	        // Check if a Controller has an error
	        #sx_ErrorActive := (#sx_ErrorController AND #iUDT_AixConfig.Motor.MotorExist)
	        OR #sFB_TimerOnOffDelayMCORunningFeedbackError.qx_DelayedSignal
	        OR #sFB_TimerOnOffDelayMCOSpeedFeedbackError.qx_DelayedSignal;

	        // Internal error
	        #sUDT_HMIStatus.InternalError := #sx_AixAvailableControler AND #sx_ErrorController;

	    END_REGION

	END_REGION

	REGION 5 - Check if configuration is ok for commissioning purposes

	    IF (
	        #iUDT_AixConfig.Motor.MotorExist                            // Check only if motor exists
	        AND (#iUDT_AixConfig.Motor.RampUpTime > 0)                  // If ramp up time is greater than 0
	        AND (#iUDT_AixConfig.Motor.RampDownTime > 0)                // and ramp down time is greater than 0
	        )
	        AND
	        (
	        #sUDT_PNDeviceController.PNDeviceFound
	        OR NOT #iUDT_AixConfig.Motor.MotorExist                       // and device found in PN structure
	        OR #ix_SimulationModeActive                                 // or simulation mode is active
	        )
	    THEN
	        #sx_ConfigurationError := FALSE;                                // Reset configuration error
	    ELSE
	        #sx_ConfigurationError := TRUE;                                 // Set configuration error
	    END_IF;

	END_REGION

	REGION 6 - Prepare output data for Controller

	    REGION 6.1 - Set direction for motor

	        // If Run forward is requested, set direction to forward
	        IF #iqUDT_ConveyorInterface.RunFwd
	            AND #iUDT_AixConfig.Motor.InterlockFwd
	        THEN
	            #sx_RunForward := TRUE;
	            #sx_RunReverse := FALSE;
	        END_IF;

	        // If Run reverse is requested, set direction into reverse
	        IF #iqUDT_ConveyorInterface.RunRvs
	            AND #iUDT_AixConfig.Motor.InterlockRvs
	        THEN
	            #sx_RunReverse := TRUE;
	            #sx_RunForward := FALSE;
	        END_IF;

	    END_REGION


	    REGION 6.3 - Stopping motor

	        // Create trigger when direction signal falling
	        #sF_TRIG_RunFwd(CLK := #iqUDT_ConveyorInterface.RunFwd);
	        #sF_TRIG_RunRvs(CLK := #iqUDT_ConveyorInterface.RunRvs);

	        // When no run signal is given the controllers should stop
	        IF (NOT #iqUDT_ConveyorInterface.RunRvs AND NOT #iqUDT_ConveyorInterface.RunFwd)
	            OR (#iqUDT_ConveyorInterface.RunRvs AND #iqUDT_ConveyorInterface.RunFwd)
	            OR (#sF_TRIG_RunRvs.Q)
	            OR (#sF_TRIG_RunFwd.Q)
	            OR #sx_ErrorActive
	        THEN
	            #sx_RunReverse := FALSE;
	            #sx_RunForward := FALSE;
	        END_IF;

	    END_REGION

	    REGION 6.5 - Check for enable operation signal

	        //Enable operation if there is no error active and there is an given direction
	        #sx_EnableOperation := NOT #sx_ErrorActive
	        AND NOT #sx_ConfigurationError
	        AND (#sx_RunForward OR #sx_RunReverse);
	    END_REGION

	    REGION 6.6 - Calculate acceleration and deceleration values

	        //Motor
	        //Recalculating Acceleration (from ms to mm)
	        #si_MotorAcceleration := REAL_TO_INT((INT_TO_REAL(#iqUDT_ConveyorInterface.SpeedSetpoint) * #iUDT_AixConfig.Motor.Ratio / 2) * (UDINT_TO_REAL(#iUDT_AixConfig.Motor.RampUpTime) / 1000));

	        //Recalculating Deceleration (from ms to mm)
	        #si_MotorDeceleration := REAL_TO_INT((INT_TO_REAL(#iqUDT_ConveyorInterface.SpeedSetpoint) * #iUDT_AixConfig.Motor.Ratio / 2) * (UDINT_TO_REAL(#iUDT_AixConfig.Motor.RampDownTime) / 1000));

	    END_REGION

	END_REGION

	REGION 7 - Write outputs to controller
	    // Clear speed setpoint when no run request or above direction request or is configuration error
	    IF #sx_EnableOperation
	    THEN
	        #sr_ActualSpeedSetpoint := INT_TO_REAL(#iqUDT_ConveyorInterface.SpeedSetpoint) / #iUDT_AixConfig.Motor.Ratio;
	    ELSE
	        #sr_ActualSpeedSetpoint := 0;
	    END_IF;

	    REGION 7.1 - Controller Left motor

	        IF #ii_MotorPositionId = #ci_Master_Left OR #ii_MotorPositionId = #ci_Slave_Left THEN
	            //Seting up speed for Left motor
	            #iqUDT_AixOutputsModule.LeftSetMotorSpeed := REAL_TO_INT(#sr_ActualSpeedSetpoint);
	            IF #iqUDT_AixOutputsModule.LeftSetMotorSpeed > #cr_MaximumOutput
	            THEN
	                // if actual value is greater than maximmu output value then write maximmu output value
	                #iqUDT_AixOutputsModule.LeftSetMotorSpeed := REAL_TO_INT(#cr_MaximumOutput);
	            END_IF;

	            //Check if motor is in use, if yes set parameters from conveyor to the controller and motor
	            IF #iUDT_AixConfig.Motor.MotorExist
	            THEN
	                //Setting up run bit, acceleration, deceleration
	                #iqUDT_AixOutputsModule.LeftMotorControl.Run := #sx_EnableOperation
	                AND (#iqUDT_ConveyorInterface.RunFwd OR #iqUDT_ConveyorInterface.RunRvs);

	                // Position setpoint
	                #iqUDT_AixOutputsModule.ServoControlDistanceLeft := #ii_PositionSetpoint;

	                //Start positioning
	                #iqUDT_AixOutputsModule.ServoControlCommandLeft.%X1 := #ix_StartPositioning
	                AND #sx_EnableOperation
	                AND (#iqUDT_ConveyorInterface.RunFwd OR #iqUDT_ConveyorInterface.RunRvs);

	                // Reset position
	                #sR_TRIG_ResetPosition(CLK := #ix_ResetPosition);

	                // Reset position after every operation
	                IF #sR_TRIG_ResetPosition.Q THEN

	                    #iqUDT_AixOutputsModule.ServoControlCommandLeft.%X0 := TRUE;

	                END_IF;

	                // End homing procedure when motor is reset
	                IF #iUDT_AixInputsModule.ServoStatusLeft.%X1 THEN

	                    #iqUDT_AixOutputsModule.ServoControlCommandLeft.%X0 := FALSE;

	                END_IF;


	                #iqUDT_AixOutputsModule.LeftSetMotorAccel := #si_MotorAcceleration;
	                #iqUDT_AixOutputsModule.LeftSetMotorDeccel := #si_MotorDeceleration;

	                //Setting direction
	                IF (#sx_RunReverse AND NOT #iUDT_AixConfig.Motor.DirectionReversal)
	                    OR (#sx_RunForward AND #iUDT_AixConfig.Motor.DirectionReversal)
	                THEN
	                    #iqUDT_AixOutputsModule.LeftMotorControl.MotorDirection := 1;
	                ELSE
	                    #iqUDT_AixOutputsModule.LeftMotorControl.MotorDirection := 0;
	                END_IF;
	            ELSE
	                #iqUDT_AixOutputsModule.LeftMotorControl.Run := FALSE;
	            END_IF;
	        END_IF;
	    END_REGION

	    REGION 7.2 - Controller right motor
	        IF #ii_MotorPositionId = #ci_Master_Right OR #ii_MotorPositionId = #ci_Slave_Right THEN
	            //Seting up speed for Right motor
	            #iqUDT_AixOutputsModule.RightSetMotorSpeed := REAL_TO_INT(#sr_ActualSpeedSetpoint);
	            IF #iqUDT_AixOutputsModule.RightSetMotorSpeed > #cr_MaximumOutput
	            THEN
	                // if actual value is greater than maximmu output value then write maximmu output value
	                #iqUDT_AixOutputsModule.RightSetMotorSpeed := REAL_TO_INT(#cr_MaximumOutput);
	            END_IF;

	            //Check if motor is in use, if yes set parameters from conveyor to the controller and motor
	            IF #iUDT_AixConfig.Motor.MotorExist
	            THEN
	                //Setting up run bit, acceleration, deceleration
	                #iqUDT_AixOutputsModule.RightMotorControl.Run := #sx_EnableOperation
	                AND (#iqUDT_ConveyorInterface.RunFwd OR #iqUDT_ConveyorInterface.RunRvs);

	                // Position setpoint
	                #iqUDT_AixOutputsModule.ServoControlDistanceRight := #ii_PositionSetpoint;

	                //Start positioning
	                #iqUDT_AixOutputsModule.ServoControlCommandRight.%X1 := #ix_StartPositioning
	                AND #sx_EnableOperation
	                AND (#iqUDT_ConveyorInterface.RunFwd OR #iqUDT_ConveyorInterface.RunRvs);

	                // Reset position
	                #sR_TRIG_ResetPosition(CLK := #ix_ResetPosition);

	                // Reset position after every operation
	                IF #sR_TRIG_ResetPosition.Q THEN

	                    #iqUDT_AixOutputsModule.ServoControlCommandRight.%X0 := TRUE;

	                END_IF;

	                // End homing procedure when motor is reset
	                IF #iUDT_AixInputsModule.ServoStatusRight.%X1 THEN

	                    #iqUDT_AixOutputsModule.ServoControlCommandRight.%X0 := FALSE;

	                END_IF;


	                #iqUDT_AixOutputsModule.RightSetMotorAccel := #si_MotorAcceleration;
	                #iqUDT_AixOutputsModule.RightSetMotorDeccel := #si_MotorDeceleration;

	                //Setting direction
	                IF (#sx_RunReverse AND NOT #iUDT_AixConfig.Motor.DirectionReversal)
	                    OR (#sx_RunForward AND #iUDT_AixConfig.Motor.DirectionReversal)
	                THEN
	                    #iqUDT_AixOutputsModule.RightMotorControl.MotorDirection := 1;
	                ELSE
	                    #iqUDT_AixOutputsModule.RightMotorControl.MotorDirection := 0;
	                END_IF;
	            ELSE
	                #iqUDT_AixOutputsModule.RightMotorControl.Run := FALSE;
	            END_IF;
	        END_IF;
	    END_REGION

	END_REGION

	REGION 8 - Reading actual speed

	    REGION 8.1 - Left Motor
	        IF #ii_MotorPositionId = #ci_Master_Left OR #ii_MotorPositionId = #ci_Slave_Left THEN
	            //When motors are in constant speed use motor actual speed
	            IF #iUDT_AixConfig.Motor.MotorExist
	            THEN
	                #si_ActualSpeed := REAL_TO_INT(INT_TO_REAL(WORD_TO_INT(#iUDT_AixInputsModule.LeftMotorActualSpeed & #cw_ActualSpeedMask)) * #iUDT_AixConfig.Motor.Ratio);
	            ELSE
	                #si_ActualSpeed := 0;
	            END_IF;
	        END_IF;
	    END_REGION

	    REGION 8.2 - Right Motor
	        IF #ii_MotorPositionId = #ci_Master_Right OR #ii_MotorPositionId = #ci_Slave_Right THEN
	            //When motors are in constant speed use motor actual speed
	            IF #iUDT_AixConfig.Motor.MotorExist
	            THEN
	                #si_ActualSpeed := REAL_TO_INT(INT_TO_REAL(WORD_TO_INT(#iUDT_AixInputsModule.RightMotorActualSpeed & #cw_ActualSpeedMask)) * #iUDT_AixConfig.Motor.Ratio);
	            ELSE
	                #si_ActualSpeed := 0;
	            END_IF;
	        END_IF;
	    END_REGION

	    REGION 8.3 - Calculation
	        //Actual speed is in mm/s
	        //Sets error signal if an motor is running for a longer time with a diferent speed than speed setpoint but after a certain time
	        #sFB_TimerOnOffDelayMCORunningFeedbackError(iudi_OnDelayTime := #cudi_FeedbackErrorDelay,
	                                                    ix_SignalToDelay := #sr_ActualSpeedSetpoint <> 0.0 AND NOT (#si_ActualSpeed <> 0));

	        //The motor should start running after specific time. If not the MCORunningFeedback error occured
	        #sFB_TimerOnOffDelayMCOSpeedFeedbackError(iudi_OnDelayTime := #cudi_FeedbackErrorDelay,
	                                                  ix_SignalToDelay := #sx_SpeedFeedbackError);

	        IF #sFB_TimerOnOffDelayMCORunningFeedbackError.qx_DelayedSignal OR #sFB_TimerOnOffDelayMCOSpeedFeedbackError.qx_DelayedSignal
	        THEN
	            #sUDT_HMIStatus.SpeedFeedbackError := TRUE;
	        END_IF;

	        //Sets signal for the time in which the motors are accelerating
	        #sFB_TimerOnOffDelayAcceleration(iudi_OnDelayTime := 0,
	                                         iudi_OffDelayTime := #iUDT_AixConfig.Motor.RampUpTime + #cudi_TimeOffsetSpeedmonitoring,
	                                         ix_SignalToDelay := #sR_TRIG_Running.Q,
	                                         ix_Enable := TRUE,
	                                         qx_DelayedSignal => #sx_Accelerating);


	        //If conveyor is running and runs forwad or backwards and is not accelerating, when any motor is running at a lower/greater speed than set speed then set an error
	        IF #iqUDT_ConveyorInterface.VFDRunning AND (#iqUDT_ConveyorInterface.RunFwd OR #iqUDT_ConveyorInterface.RunRvs) AND NOT #sx_Accelerating
	        THEN
	            //Check if the difference betwen acctual speed and set speed is bigger than deviation then set error
	            #sx_SpeedFeedbackError := #iUDT_AixConfig.Motor.SpeedSetpointWindow < (ABS(#si_ActualSpeed) - (#iqUDT_ConveyorInterface.SpeedSetpoint));
	        END_IF;


	        // Check IF speed setpoint is reached FOR motor
	        #sx_SpeedSetpointReached := (ABS(#si_ActualSpeed) >= ((#iqUDT_ConveyorInterface.SpeedSetpoint) - #iUDT_AixConfig.Motor.SpeedSetpointWindow))
	        AND (ABS(#si_ActualSpeed) <= ((#iqUDT_ConveyorInterface.SpeedSetpoint) + #iUDT_AixConfig.Motor.SpeedSetpointWindow));
	    END_REGION

	END_REGION

	(* REGION 9 - Reading actual position

	    REGION 9.1 - Left Motor

	        #sx_LeftServoHomeHasBeenSet := #iUDT_AixInputsModule.ServoStatusLeft.%X1;
	        IF #ix_MotorPositionId = #ci_Left
	        THEN
	            IF #sx_LeftServoHomeHasBeenSet THEN
	                #si_LastLeftMotorPosition := 0;
	            END_IF;
	            // Add last position change to static memory
	            #si_LeftMotorPosition += - #si_LastLeftMotorPosition;
	            // Save last motor position
	            #si_LastLeftMotorPosition := #iUDT_AixInputsModule.ServoLocationLeft;

	            // Copy displacement if motor position change is greater or equal to 1 cm and store rest
	            IF #si_LeftMotorPosition > 10 THEN
	                #iqUDT_ConveyorInterface.DeltaPosition := REAL_TO_INT(INT_TO_REAL(#si_LeftMotorPosition) * #iUDT_AixConfig.Motor.Ratio) / 10;
	                #si_LeftMotorPosition := #si_LeftMotorPosition MOD 10;
	            ELSE
	                #iqUDT_ConveyorInterface.DeltaPosition := 0;
	            END_IF;

	            // allocate Motor Rotation status
	            #sb_MotorRotationStatus.%X0 := #iUDT_AixInputsModule.LeftMotorDiagnostic.MotorStatus1;
	            #sb_MotorRotationStatus.%X1 := #iUDT_AixInputsModule.LeftMotorDiagnostic.MotorStatus2;

	            // Change direction sign if motor running reverse
	            IF ((#sb_MotorRotationStatus = #cb_MotorInCW) AND NOT #iUDT_AixConfig.Motor.DirectionReversal) OR
	                ((#sb_MotorRotationStatus = #cb_MotorInCCW) AND #iUDT_AixConfig.Motor.DirectionReversal)
	            THEN

	                #iqUDT_ConveyorInterface.DeltaPosition *= -1;

	            END_IF;

	            // Motor positioned
	            #qx_Positioned := #iUDT_AixInputsModule.ServoStatusLeft.%X0;

	        END_IF;

	    END_REGION

	    REGION 9.2 - Right motor
	        #sx_RightServoHomeHasBeenSet := #iUDT_AixInputsModule.ServoStatusRight.%X1;
	        IF #ix_MotorPositionId = #ci_Right
	        THEN
	            IF #sx_RightServoHomeHasBeenSet THEN
	                #si_LastRightMotorPosition := 0;
	            END_IF;
	            // Add last position change to static memory
	            #si_RightMotorPosition += - #si_LastRightMotorPosition;
	            // Save last motor position
	            #si_LastRightMotorPosition := #iUDT_AixInputsModule.ServoLocationRight;

	            // Copy displacement if motor position change is greater or equal to 1 cm and store rest
	            IF #si_RightMotorPosition > 10 THEN
	                #iqUDT_ConveyorInterface.DeltaPosition := REAL_TO_INT(INT_TO_REAL(#si_RightMotorPosition) * #iUDT_AixConfig.Motor.Ratio) / 10;
	                #si_RightMotorPosition := #si_RightMotorPosition MOD 10;
	            ELSE
	                #iqUDT_ConveyorInterface.DeltaPosition := 0;
	            END_IF;

	            // allocate Motor Rotation status
	            #sb_MotorRotationStatus.%X0 := #iUDT_AixInputsModule.RightMotorDiagnostic.MotorStatus1;
	            #sb_MotorRotationStatus.%X1 := #iUDT_AixInputsModule.RightMotorDiagnostic.MotorStatus2;

	            // Change direction sign if motor running reverse
	            IF ((#sb_MotorRotationStatus = #cb_MotorInCW) AND NOT #iUDT_AixConfig.Motor.DirectionReversal) OR
	                ((#sb_MotorRotationStatus = #cb_MotorInCCW) AND #iUDT_AixConfig.Motor.DirectionReversal)
	            THEN

	                #iqUDT_ConveyorInterface.DeltaPosition *= -1;

	            END_IF;

	            // Motor positioned
	            #qx_Positioned := #iUDT_AixInputsModule.ServoStatusRight.%X0;

	        END_IF;

	    END_REGION


	END_REGION *)

	REGION 9 - Reading actual position

	    REGION 9.1 - Left motor

	        IF #ii_MotorPositionId = #ci_Master_Left OR #ii_MotorPositionId = #ci_Slave_Left
	        THEN
	            IF #iUDT_AixInputsModule.ServoLocationLeft = 0 THEN
	                #si_LastLeftMotorPosition := 0;
	            END_IF;
	            // Add last position change to static memory
	            #si_LeftMotorPosition += ABS(ABS(#iUDT_AixInputsModule.ServoLocationLeft) - ABS(#si_LastLeftMotorPosition));
	            // Save last motor position
	            #si_LastLeftMotorPosition := #iUDT_AixInputsModule.ServoLocationLeft;

	            // Copy delta position if motor position change is greater or equal to 1 cm and store rest
	            IF #si_LeftMotorPosition > 10 THEN
	                IF #ii_MotorPositionId = #ci_Master_Left THEN
	                    #iqUDT_ConveyorInterface.DeltaPosition := REAL_TO_INT(INT_TO_REAL(#si_LeftMotorPosition) * #iUDT_AixConfig.Motor.Ratio) / 10;
	                END_IF;
	                #si_LeftMotorPosition := #si_LeftMotorPosition MOD 10;
	            ELSE
	                IF #ii_MotorPositionId = #ci_Master_Left THEN
	                    #iqUDT_ConveyorInterface.DeltaPosition := 0;
	                END_IF;
	            END_IF;
	            // Change direction sign if motor running reverse
	            IF #iUDT_AixInputsModule.LeftMotorDiagnostic.MotorStatus1 AND NOT #iUDT_AixInputsModule.LeftMotorDiagnostic.MotorStatus2 AND NOT #iUDT_AixConfig.Motor.DirectionReversal
	                OR NOT #iUDT_AixInputsModule.LeftMotorDiagnostic.MotorStatus1 AND #iUDT_AixInputsModule.LeftMotorDiagnostic.MotorStatus2 AND #iUDT_AixConfig.Motor.DirectionReversal
	            THEN
	                IF #ii_MotorPositionId = #ci_Master_Left THEN
	                    #iqUDT_ConveyorInterface.DeltaPosition *= -1;
	                END_IF;
	            END_IF;

	            // Motor positioned
	            #qx_Positioned := #iUDT_AixInputsModule.ServoStatusLeft.%X0;

	        END_IF;

	    END_REGION

	    REGION 9.2 - Right motor

	        IF #ii_MotorPositionId = #ci_Master_Right OR #ii_MotorPositionId = #ci_Slave_Right
	        THEN
	            IF #iUDT_AixInputsModule.ServoLocationRight = 0 THEN
	                #si_LastRightMotorPosition := 0;
	            END_IF;
	            // Add last position change to static memory
	            #si_RightMotorPosition += ABS(ABS(#iUDT_AixInputsModule.ServoLocationRight) - ABS(#si_LastRightMotorPosition));
	            // Save last motor position
	            #si_LastRightMotorPosition := #iUDT_AixInputsModule.ServoLocationRight;

	            // Copy delta position if motor position change is greater or equal to 1 cm and store rest
	            IF #si_RightMotorPosition > 10 THEN
	                IF #ii_MotorPositionId = #ci_Master_Right THEN
	                    #iqUDT_ConveyorInterface.DeltaPosition := REAL_TO_INT(INT_TO_REAL(#si_RightMotorPosition) * #iUDT_AixConfig.Motor.Ratio) / 10;
	                END_IF;
	                #si_RightMotorPosition := #si_RightMotorPosition MOD 10;
	            ELSE
	                IF #ii_MotorPositionId = #ci_Master_Right THEN
	                    #iqUDT_ConveyorInterface.DeltaPosition := 0;
	                END_IF;
	            END_IF;
	            // Change direction sign if motor running reverse
	            IF #iUDT_AixInputsModule.RightMotorDiagnostic.MotorStatus1 AND NOT #iUDT_AixInputsModule.RightMotorDiagnostic.MotorStatus2 AND NOT #iUDT_AixConfig.Motor.DirectionReversal
	                OR NOT #iUDT_AixInputsModule.RightMotorDiagnostic.MotorStatus1 AND #iUDT_AixInputsModule.RightMotorDiagnostic.MotorStatus2 AND #iUDT_AixConfig.Motor.DirectionReversal
	            THEN
	                IF #ii_MotorPositionId = #ci_Master_Right THEN
	                    #iqUDT_ConveyorInterface.DeltaPosition *= -1;
	                END_IF;
	            END_IF;

	            // Motor positioned
	            #qx_Positioned := #iUDT_AixInputsModule.ServoStatusRight.%X0;

	        END_IF;

	    END_REGION

	END_REGION


	REGION 10 - Copy signals to interface DB and to status output UDT

	    REGION 10.1 - Motor

	        // Create internal error status
	        // Write Conveyor interface bits only if it is a Master
	        IF #ii_MotorPositionId = #ci_Master_Left OR #ii_MotorPositionId = #ci_Master_Right THEN

	            #iqUDT_ConveyorInterface.VFDRunning := #sx_AixAvailableControler AND
	            (#si_ActualSpeed <> 0);                 // Write true on output Conveyor interface structure if Ai2's are in operation and motor is turning

	            #iqUDT_ConveyorInterface.VFDatSpeed := #sx_SpeedSetpointReached AND
	            #sx_AixAvailableControler AND
	            #si_ActualSpeed <> 0 AND
	            NOT #sx_SpeedFeedbackError;             // Copy setpoint speed reached state from static to the output conveyor interface structure

	            #iqUDT_ConveyorInterface.InternalWarningVFD := #sUDT_HMIStatus.PNSlaveWarning;                                                       // Set the internal warning bit if any warning is active

	            #iqUDT_ConveyorInterface.InternalErrorVFD := #sx_ErrorCMotor;                   // Set the internal error bit if any fault is active

	            #iqUDT_ConveyorInterface.ActualSpeed := ABS(#si_ActualSpeed);                   // Copy the calculated value to the output

	            #iqUDT_ConveyorInterface.ConfigurationError := #sx_ConfigurationError;          // Copy the calculated value to the output

	        END_IF;


	    END_REGION

	    REGION 10.2 - Move error status TO HMI Status

	        // Copy error status to output
	        #qUDT_HMIStatus := #sUDT_HMIStatus;

	    END_REGION

	END_REGION

	REGION 11 - Statistic

	    REGION 11.1 - General
	        // Statement section REGION
	        #sx_GeneralStatisticsReset := #iqUDT_ConveyorInterface.ResetStatistics;
	    END_REGION

	    // Create trigger on error and create statistics for profinet slave not online
	    #sR_TRIG_PNSlaveNotOnline(CLK := #sUDT_HMIStatus.PNSlaveNotOnline);                 // Detect the rising edge of the error

	    IF #sx_GeneralStatisticsReset OR #sUDT_HMIStatus.PNSlaveNotOnline
	    THEN

	        "FC_Statistics"(ix_Reset := #sx_GeneralStatisticsReset,
	                        ix_Activate := #sUDT_HMIStatus.PNSlaveNotOnline,
	                        ix_RTrigActivate := #sR_TRIG_PNSlaveNotOnline.Q,
	                        iqUDT_Statistics := #iqUDT_MCOStatistics.PNSlaveNotOnline);

	        #iqUDT_MCOStatistics.PNSlaveNotOnline := #iqUDT_MCOStatistics.PNSlaveNotOnline;
	    END_IF;

	    // Create trigger on error and create statistics for profinet slave error
	    #sR_TRIG_PNSlaveError(CLK := #sUDT_HMIStatus.PNSlaveError);                                                                          // Detect the rising edge of the error

	    IF #sx_GeneralStatisticsReset OR #sUDT_HMIStatus.PNSlaveError
	    THEN

	        "FC_Statistics"(ix_Reset := #sx_GeneralStatisticsReset,
	                        ix_Activate := #sUDT_HMIStatus.PNSlaveError,
	                        ix_RTrigActivate := #sR_TRIG_PNSlaveError.Q,
	                        iqUDT_Statistics := #iqUDT_MCOStatistics.PNSlaveError);

	        #iqUDT_MCOStatistics.PNSlaveError := #iqUDT_MCOStatistics.PNSlaveError;
	    END_IF;


	    // Create trigger on error and create statistics for MCO communication error
	    #sR_TRIG_CommunicationErrorMCO(CLK := #qUDT_HMIStatus.CommunicationErrorVFD);            // Detect the rising edge of the error

	    IF #sx_GeneralStatisticsReset OR #qUDT_HMIStatus.CommunicationErrorVFD
	    THEN

	        "FC_Statistics"(ix_Reset := #sx_GeneralStatisticsReset,
	                        ix_Activate := #qUDT_HMIStatus.CommunicationErrorVFD,
	                        ix_RTrigActivate := #sR_TRIG_CommunicationErrorMCO.Q,
	                        iqUDT_Statistics := #iqUDT_MCOStatistics.CommunicationErrorMovikit);

	    END_IF;

	    REGION 11.1 - Motor

	        // Create trigger on error and create statistics for internal MCO Error
	        #sR_TRIG_MCOInternalError(CLK := #sUDT_HMIStatus.InternalError);         // Detect the rising edge of the error

	        IF #iqUDT_ConveyorInterface.ResetStatistics OR #sUDT_HMIStatus.InternalError
	        THEN

	            "FC_Statistics"(ix_Reset := #iqUDT_ConveyorInterface.ResetStatistics,
	                            ix_Activate := #sUDT_HMIStatus.InternalError,
	                            ix_RTrigActivate := #sR_TRIG_MCOInternalError.Q,
	                            iqUDT_Statistics := #iqUDT_MCOStatistics.VFDInternalError);

	        END_IF;

	        // Create trigger on running signal and create statistics for running status
	        #sR_TRIG_Running(CLK := #iqUDT_ConveyorInterface.VFDRunning);                           // Detect the rising edge of the signal

	        IF #iqUDT_ConveyorInterface.ResetStatistics OR #iqUDT_ConveyorInterface.VFDRunning
	        THEN

	            "FC_Statistics"(ix_Reset := #iqUDT_ConveyorInterface.ResetStatistics,
	                            ix_Activate := #iqUDT_ConveyorInterface.VFDRunning,
	                            ix_RTrigActivate := #sR_TRIG_Running.Q,
	                            iqUDT_Statistics := #iqUDT_MCOStatistics.Running);
	        END_IF;


	    END_REGION
	    REGION 12 Status bit allocation
	        "FC_BitAllocation"(ix_Bit0 := #qUDT_HMIStatus.SpeedFeedbackError,
	                           ix_Bit1 := #qUDT_HMIStatus.InternalWarning,
	                           ix_Bit2 := #qUDT_HMIStatus.InternalError,
	                           ix_Bit3 := #qUDT_HMIStatus.CommunicationErrorVFD,
	                           ix_Bit4 := #qUDT_HMIStatus.PNSlaveNotOnline,
	                           ix_Bit5 := #qUDT_HMIStatus.PNSlaveError,
	                           ix_Bit6 := #qUDT_HMIStatus.PNSlaveWarning,
	                           ix_Bit7 := FALSE,
	                           ix_Bit8 := FALSE,
	                           ix_Bit9 := FALSE,
	                           ix_Bit10 := FALSE,
	                           ix_Bit11 := FALSE,
	                           ix_Bit12 := FALSE,
	                           ix_Bit13 := FALSE,
	                           ix_Bit14 := FALSE,
	                           ix_Bit15 := FALSE,
	                           ix_Bit16 := FALSE,
	                           ix_Bit17 := FALSE,
	                           ix_Bit18 := FALSE,
	                           ix_Bit19 := FALSE,
	                           ix_Bit20 := FALSE,
	                           ix_Bit21 := FALSE,
	                           ix_Bit22 := FALSE,
	                           ix_Bit23 := FALSE,
	                           ix_Bit24 := FALSE,
	                           ix_Bit25 := FALSE,
	                           ix_Bit26 := FALSE,
	                           ix_Bit27 := FALSE,
	                           ix_Bit28 := FALSE,
	                           ix_Bit29 := FALSE,
	                           ix_Bit30 := FALSE,
	                           ix_Bit31 := FALSE,
	                           qdw_Dword => #qUDT_HMIStatus.ControllerStatus);
	    END_REGION
	END_REGION
END_FUNCTION_BLOCK

FUNCTION_BLOCK "FB_Displacement"
TITLE = FB_Displacement
{ S7_Optimized_Access := 'TRUE' }
AUTHOR : MHSE
FAMILY : GeneralSystemFunctions
VERSION : 3.0
//Function block to calculate the displacement.
   VAR_IN_OUT
      iqUDT_ConveyorInterface : "UDT_ConveyorInterface";   // Conveyor interface structure Motor
   END_VAR

   VAR
      slr_FormDisplacement { ExternalAccessible := 'False'; ExternalVisible := 'False'; ExternalWritable := 'False'} : LReal;   // Conveyor displacement [cm]
      slr_Correction { ExternalAccessible := 'False'; ExternalVisible := 'False'; ExternalWritable := 'False'} : LReal;   // Correction [cm]
      sx_PositionModeActive { ExternalAccessible := 'False'; ExternalVisible := 'False'; ExternalWritable := 'False'} : Bool;   // Position Mode is used, Will reset after power change
   END_VAR

   VAR_TEMP
      ti_Displacement : Int;   // Conveyor displacement [cm]
   END_VAR

   VAR CONSTANT
      ci_IntMin : Int := -32768;
      ci_IntMax : Int := 32767;
   END_VAR


BEGIN
	(*
	----------------------------------------------------------------------------------------

	Version history:
	Date        | Version   | Author        | Remark
	----------------------------------------------------------------------------------------
	24/05/2019  | 0.1       | L.Klar        | first release MHS TIA 15.1
	24/07/2019  | 2.0       | L.Klar        | 2.0 MHS library release TIA 15.1
	12/09/2019  | 2.1       | P.Majka       | Comments updataed
	04/11/2019  | 2.2       | L.Klar        | Prevoius cycle scan changed from memory to DB variable
	12/11/2019  | 3.0       | P.Majka       | 3.0 MHS library release TIA 15.1
	21/02/2023  | 4.0       | F.Baten       | 4.0 Release TIA 17.5
	31/05/2024  | 4.1       | I.Ajram       | Added Displacement from Position feedback
	*)
	REGION 0 - Mode detection
	    IF #iqUDT_ConveyorInterface.DeltaPosition <> 0 THEN
	        #sx_PositionModeActive := true;
	    END_IF;
	END_REGION


	REGION 1 - Displacement From Speed
	    IF NOT #sx_PositionModeActive THEN
	        REGION 1.1 Calculate Displacement
	            // Displacement is calculated using actual conveyor speed and the previous PLC cycle scan time
	            #slr_FormDisplacement := INT_TO_LREAL(#iqUDT_ConveyorInterface.ActualSpeed) * "DB_Memory".PrevCycleTime / 10000.0;

	            // Correction is used to accumulate the rest of the calculated value
	            #slr_Correction := FRAC(#slr_FormDisplacement) + #slr_Correction;

	            // The actual displacement is a sum of complete parts of the displacement and correction variables
	            #ti_Displacement := DINT_TO_INT(TRUNC(#slr_FormDisplacement) + TRUNC(#slr_Correction));

	        END_REGION

	        REGION 1.2 - Correction check

	            // Correction incrementation or decremantation if it exceeds 1 or -1 in case of negative speed
	            IF (#slr_Correction >= 1)
	            THEN

	                #slr_Correction -= 1;

	            ELSIF (#slr_Correction <= -1)
	            THEN

	                #slr_Correction += 1;

	            END_IF;

	        END_REGION

	        #iqUDT_ConveyorInterface.Displacement := #ti_Displacement;
	    END_IF;
	END_REGION

	REGION 2 - Displacement from Position
	    // pass position displacement from Servo Feedback
	    IF #sx_PositionModeActive THEN
	        #iqUDT_ConveyorInterface.Displacement := #iqUDT_ConveyorInterface.DeltaPosition;

	    END_IF;

	END_REGION
END_FUNCTION_BLOCK

FUNCTION_BLOCK "FB_RightAngledTransfer"
{ S7_Optimized_Access := 'TRUE' }
VERSION : 0.1
   VAR_INPUT
      iUDT_Configuration { ExternalAccessible := 'False'; ExternalVisible := 'False'; ExternalWritable := 'False'} : "UDT_RATConfiguration" := ((), (), (), (), (), (), (), (), (), (), (), (), (), (), 1, 2, 3, 4, (), (), (), ());   // Configuration structure
      iUDT_LowerConveyorConfiguration { ExternalAccessible := 'False'; ExternalVisible := 'False'; ExternalWritable := 'False'} : "UDT_ConveyorConfiguration";   // Lower configuration structure
      iUDT_UpperConveyorConfiguration { ExternalAccessible := 'False'; ExternalVisible := 'False'; ExternalWritable := 'False'} : "UDT_ConveyorConfiguration";   // Upper configuration structure
      iUDT_PECConfiguration { ExternalAccessible := 'False'; ExternalVisible := 'False'; ExternalWritable := 'False'} : "UDT_PECConfiguration";   // PEC configuration structure
      ii_DestinationA { ExternalAccessible := 'False'; ExternalVisible := 'False'; ExternalWritable := 'False'} : Int;   // Forced destination for every product from conveyor A. When this is 0 then destination is taken from GIN
      ii_DestinationB { ExternalAccessible := 'False'; ExternalVisible := 'False'; ExternalWritable := 'False'} : Int;   // Forced destination for every product from conveyor B. When this is 0 then destination is taken from GIN
      ii_DestinationC { ExternalAccessible := 'False'; ExternalVisible := 'False'; ExternalWritable := 'False'} : Int;   // Forced destination for every product from conveyor C. When this is 0 then destination is taken from GIN
      ii_DestinationD { ExternalAccessible := 'False'; ExternalVisible := 'False'; ExternalWritable := 'False'} : Int;   // Forced destination for every product from conveyor D. When this is 0 then destination is taken from GIN
      ix_HardwareOk { ExternalAccessible := 'False'; ExternalVisible := 'False'; ExternalWritable := 'False'} : Bool;   // TRUE when  hardware is Ok
      ix_400vOk { ExternalAccessible := 'False'; ExternalVisible := 'False'; ExternalWritable := 'False'} : Bool;   // TRUE when 400VAC is healthy
      ix_24vOk { ExternalAccessible := 'False'; ExternalVisible := 'False'; ExternalWritable := 'False'} : Bool;   // TRUE when 24VDC is healthy
      ix_SafetyOk { ExternalAccessible := 'False'; ExternalVisible := 'False'; ExternalWritable := 'False'} : Bool;   // TRUE when safety is ok
      ix_AirPressureOk { ExternalAccessible := 'False'; ExternalVisible := 'False'; ExternalWritable := 'False'} : Bool;   // Air pressure circuit healthy
      ix_SectionIsDown { ExternalAccessible := 'False'; ExternalVisible := 'False'; ExternalWritable := 'False'} : Bool;   // TRUE when section is down
      ix_SectionIsUp { ExternalAccessible := 'False'; ExternalVisible := 'False'; ExternalWritable := 'False'} : Bool;   // TRUE when section is up
      ix_ConveyorAAuto { ExternalAccessible := 'False'; ExternalVisible := 'False'; ExternalWritable := 'False'} : Bool;   // Conveyor is started in auto
      ix_ConveyorBAuto { ExternalAccessible := 'False'; ExternalVisible := 'False'; ExternalWritable := 'False'} : Bool;   // Conveyor is started in auto
      ix_ConveyorCAuto { ExternalAccessible := 'False'; ExternalVisible := 'False'; ExternalWritable := 'False'} : Bool;   // Conveyor is started in auto
      ix_ConveyorDAuto { ExternalAccessible := 'False'; ExternalVisible := 'False'; ExternalWritable := 'False'} : Bool;   // Conveyor is started in auto
      ix_PEC { ExternalAccessible := 'False'; ExternalVisible := 'False'; ExternalWritable := 'False'} : Bool;   // True when outfeed PEC is not occupied
      ix_ExternalReceiveRequestA { ExternalAccessible := 'False'; ExternalVisible := 'False'; ExternalWritable := 'False'} : Bool;   // Send parcel request from A conveyor
      ix_ExternalReceiveRequestB { ExternalAccessible := 'False'; ExternalVisible := 'False'; ExternalWritable := 'False'} : Bool;   // Send parcel request from B conveyor
      ix_ExternalReceiveRequestC { ExternalAccessible := 'False'; ExternalVisible := 'False'; ExternalWritable := 'False'} : Bool;   // Send parcel request from C conveyor
      ix_ExternalReceiveRequestD { ExternalAccessible := 'False'; ExternalVisible := 'False'; ExternalWritable := 'False'} : Bool;   // Send parcel request from D conveyor
      ix_PECInfeedA { ExternalAccessible := 'False'; ExternalVisible := 'False'; ExternalWritable := 'False'} : Bool;   // End of section from infeed A
      ix_PECInfeedB { ExternalAccessible := 'False'; ExternalVisible := 'False'; ExternalWritable := 'False'} : Bool;   // End of section from infeed B
      ix_PECInfeedC { ExternalAccessible := 'False'; ExternalVisible := 'False'; ExternalWritable := 'False'} : Bool;   // End of section from infeed C
      ix_PECInfeedD { ExternalAccessible := 'False'; ExternalVisible := 'False'; ExternalWritable := 'False'} : Bool;   // End of section from infeed D
   END_VAR

   VAR_OUTPUT
      qUDT_HMIRATStatus { ExternalAccessible := 'False'; ExternalVisible := 'False'; ExternalWritable := 'False'} : "UDT_RATStatus";   // HMI status structure
      qUDT_HMIConveyorStatus { ExternalAccessible := 'False'; ExternalVisible := 'False'; ExternalWritable := 'False'} : "UDT_ConveyorStatus";   // HMI status structure for lower conveyor
      qUDT_HMIPECStatus { ExternalAccessible := 'False'; ExternalVisible := 'False'; ExternalWritable := 'False'} : "UDT_PECStatus";   // HMI status structure for PEC
      qUDT_RATStatus { ExternalAccessible := 'False'; ExternalVisible := 'False'; ExternalWritable := 'False'} : "UDT_CommonStatus";   // Common status structure
      qUDT_ConveyorStatus { ExternalAccessible := 'False'; ExternalVisible := 'False'; ExternalWritable := 'False'} : "UDT_CommonStatus";   // Common status structure for lower conveyor
      qx_PopupControl { ExternalAccessible := 'False'; ExternalVisible := 'False'; ExternalWritable := 'False'} : Bool;   // Output to control popup section
      qx_ExternalSendRequestA { ExternalAccessible := 'False'; ExternalVisible := 'False'; ExternalWritable := 'False'} : Bool;   // Send request to next RAT in A direction
      qx_ExternalSendRequestB { ExternalAccessible := 'False'; ExternalVisible := 'False'; ExternalWritable := 'False'} : Bool;   // Send request to next RAT in B direction
      qx_ExternalSendRequestC { ExternalAccessible := 'False'; ExternalVisible := 'False'; ExternalWritable := 'False'} : Bool;   // Send request to next RAT in C direction
      qx_ExternalSendRequestD { ExternalAccessible := 'False'; ExternalVisible := 'False'; ExternalWritable := 'False'} : Bool;   // Send request to next RAT in D direction
   END_VAR

   VAR_IN_OUT
      iqUDT_EquipmentControl : "UDT_EquipmentControl";   // Equipment control structure
      iqUDT_RATCommand : "UDT_RATCommand";   // RAT command stucture
      iqUDT_ConveyorCommand : "UDT_ConveyorCommand";   // Conveyor command stucture
      iqUDT_RATStatistics : "UDT_RATStatistics";   // RAT statistics structure
      iqUDT_ConveyorStatistics : "UDT_ConveyorStatistics";   // Statistics structure
      iqUDT_PECStatistics : "UDT_PECStatistics";   // PEC statistics structure
      iqUDT_HandShakeConveyorA : "UDT_ConveyorHandshake";   // Handshake structure low level conveyor
      iqUDT_HandShakeConveyorB : "UDT_ConveyorHandshake";   // Handshake structure low level conveyor
      iqUDT_HandShakeConveyorC : "UDT_ConveyorHandshake";   // Handshake structure high level conveyor
      iqUDT_HandShakeConveyorD : "UDT_ConveyorHandshake";   // Handshake structure high level conveyor
      iqUDT_LowerConveyorInterface : "UDT_ConveyorInterface";   // Lower conveyor interface structure
      iqUDT_UpperConveyorInterface : "UDT_ConveyorInterface";   // Upper conveyor interface structure
      iqUDT_RATPositioning : "UDT_RATPositioning";   // Positioning control structure
      iqUDT_BladeStopEoSInterface : "UDT_ValveInterface";   // Blade stop EoS interface signals
      iqUDT_BladeStopBoSInterface : "UDT_ValveInterface";   // Blade stop BoS interface signals
   END_VAR

   VAR RETAIN
      sa_FiFo { ExternalAccessible := 'False'; ExternalVisible := 'False'; ExternalWritable := 'False'} : Array[1..#ci_FiFoLength] of Int := [10(0)];   // FiFo of request
   END_VAR
   VAR
      sUDT_CommonStatus { ExternalAccessible := 'False'; ExternalVisible := 'False'; ExternalWritable := 'False'; S7_SetPoint := 'False'} : "UDT_CommonStatus";   // Common status structure
      sUDT_HMIStatus { ExternalAccessible := 'False'; ExternalVisible := 'False'; ExternalWritable := 'False'; S7_SetPoint := 'False'} : "UDT_RATStatus";   // HMI status structure
      sUDT_HandshakeBuffer { ExternalAccessible := 'False'; ExternalVisible := 'False'; ExternalWritable := 'False'; S7_SetPoint := 'False'} : "UDT_ConveyorHandshake";   // Auxiliary handshake structure
      sUDT_HandshakeUpLowerConveyor { ExternalAccessible := 'False'; ExternalVisible := 'False'; ExternalWritable := 'False'; S7_SetPoint := 'False'} : "UDT_ConveyorHandshake";   // Upstream handshake for lower conveyor
      sUDT_HandshakeUpUpperConveyor { ExternalAccessible := 'False'; ExternalVisible := 'False'; ExternalWritable := 'False'; S7_SetPoint := 'False'} : "UDT_ConveyorHandshake";   // Upstream handshake for upper conveyor
      sUDT_HandshakeLowerConveyor { ExternalAccessible := 'False'; ExternalVisible := 'False'; ExternalWritable := 'False'; S7_SetPoint := 'False'} : "UDT_ConveyorHandshake";   // Downstream handshake for lower conveyor
      sUDT_HandshakeUpperConveyor { ExternalAccessible := 'False'; ExternalVisible := 'False'; ExternalWritable := 'False'; S7_SetPoint := 'False'} : "UDT_ConveyorHandshake";   // Downstream handshake for upper conveyor
      sFB_Conveyor_LowerConveyor { ExternalAccessible := 'False'; ExternalVisible := 'False'; ExternalWritable := 'False'; S7_SetPoint := 'False'} : "FB_Conveyor";   // Lower conveyor block instance
      sFB_Conveyor_UpperConveyor { ExternalAccessible := 'False'; ExternalVisible := 'False'; ExternalWritable := 'False'; S7_SetPoint := 'False'} : "FB_Conveyor";   // Upper conveyor block instance
      sFB_SectionUpMonitor { ExternalAccessible := 'False'; ExternalVisible := 'False'; ExternalWritable := 'False'; S7_SetPoint := 'False'} : "FB_TimerOnOffDelay";   // Timer to monitor divert took too long to move to upper position
      sFB_SectionDownMonitor { ExternalAccessible := 'False'; ExternalVisible := 'False'; ExternalWritable := 'False'; S7_SetPoint := 'False'} : "FB_TimerOnOffDelay";   // Timer to monitor divert took too long to move to lower position
      sFB_PECOnOffDelay { ExternalAccessible := 'False'; ExternalVisible := 'False'; ExternalWritable := 'False'; S7_SetPoint := 'False'} : "FB_TimerOnOffDelay";   // Timer for PEC filtering
      sFB_InfeedTimeout { ExternalAccessible := 'False'; ExternalVisible := 'False'; ExternalWritable := 'False'; S7_SetPoint := 'False'} : "FB_TimerOnOffDelay";   // Timer to monitor infeed timeout
      sFB_ConveyorAReactivation { ExternalAccessible := 'False'; ExternalVisible := 'False'; ExternalWritable := 'False'; S7_SetPoint := 'False'} : "FB_TimerOnOffDelay";   // Timer to monitor reativation on Conveyor A
      sFB_ConveyorBReactivation { ExternalAccessible := 'False'; ExternalVisible := 'False'; ExternalWritable := 'False'; S7_SetPoint := 'False'} : "FB_TimerOnOffDelay";   // Timer to monitor reativation on Conveyor B
      sFB_ConveyorCReactivation { ExternalAccessible := 'False'; ExternalVisible := 'False'; ExternalWritable := 'False'; S7_SetPoint := 'False'} : "FB_TimerOnOffDelay";   // Timer to monitor reativation on Conveyor C
      sFB_ConveyorDReactivation { ExternalAccessible := 'False'; ExternalVisible := 'False'; ExternalWritable := 'False'; S7_SetPoint := 'False'} : "FB_TimerOnOffDelay";   // Timer to monitor reativation on Conveyor D
      sFB_PEC { ExternalAccessible := 'False'; ExternalVisible := 'False'; ExternalWritable := 'False'; S7_SetPoint := 'False'} : "FB_PEC";   // RAT PEC handling
      sR_TRIG_ReceiveRequestConveyorA {InstructionName := 'R_TRIG'; LibVersion := '1.0'; ExternalAccessible := 'False'; ExternalVisible := 'False'; ExternalWritable := 'False'; S7_SetPoint := 'False'} : R_TRIG;   // Rising edge trigger RTS signal from infeed
      sR_TRIG_ReceiveRequestConveyorB {InstructionName := 'R_TRIG'; LibVersion := '1.0'; ExternalAccessible := 'False'; ExternalVisible := 'False'; ExternalWritable := 'False'; S7_SetPoint := 'False'} : R_TRIG;   // Rising edge trigger RTS signal from infeed
      sR_TRIG_ReceiveRequestConveyorC {InstructionName := 'R_TRIG'; LibVersion := '1.0'; ExternalAccessible := 'False'; ExternalVisible := 'False'; ExternalWritable := 'False'; S7_SetPoint := 'False'} : R_TRIG;   // Rising edge trigger RTS signal from infeed
      sR_TRIG_ReceiveRequestConveyorD {InstructionName := 'R_TRIG'; LibVersion := '1.0'; ExternalAccessible := 'False'; ExternalVisible := 'False'; ExternalWritable := 'False'; S7_SetPoint := 'False'} : R_TRIG;   // Rising edge trigger RTS signal from infeed
      sR_TRIG_ManualMode {InstructionName := 'R_TRIG'; LibVersion := '1.0'; ExternalAccessible := 'False'; ExternalVisible := 'False'; ExternalWritable := 'False'; S7_SetPoint := 'False'} : R_TRIG;   // Rising edge trigger manual mode
      sF_TRIG_ManualMode {InstructionName := 'F_TRIG'; LibVersion := '1.0'; ExternalAccessible := 'False'; ExternalVisible := 'False'; ExternalWritable := 'False'; S7_SetPoint := 'False'} : F_TRIG;   // Falling edge trigger manual mode
      sR_TRIG_ManualGoUp {InstructionName := 'R_TRIG'; LibVersion := '1.0'; ExternalAccessible := 'False'; ExternalVisible := 'False'; ExternalWritable := 'False'; S7_SetPoint := 'False'} : R_TRIG;   // Rising edge run conveyor in manual mode
      sR_TRIG_ManualGoDown {InstructionName := 'R_TRIG'; LibVersion := '1.0'; ExternalAccessible := 'False'; ExternalVisible := 'False'; ExternalWritable := 'False'; S7_SetPoint := 'False'} : R_TRIG;   // Rising edge trigger manual jog
      sR_TRIG_PecOutfeed {InstructionName := 'R_TRIG'; LibVersion := '1.0'; ExternalAccessible := 'False'; ExternalVisible := 'False'; ExternalWritable := 'False'; S7_SetPoint := 'False'} : R_TRIG;   // Rising edge of reverse direction
      sF_TRIG_Jog {InstructionName := 'F_TRIG'; LibVersion := '1.0'; ExternalAccessible := 'False'; ExternalVisible := 'False'; ExternalWritable := 'False'; S7_SetPoint := 'False'} : F_TRIG;   // Falling edge trigger manual mode jog
      sR_TRIG_LowerInfeed {InstructionName := 'R_TRIG'; LibVersion := '1.0'; ExternalAccessible := 'False'; ExternalVisible := 'False'; ExternalWritable := 'False'; S7_SetPoint := 'False'} : R_TRIG;   // Rising edge of infeeding on lower conveyor
      sR_TRIG_UpperInfeed {InstructionName := 'R_TRIG'; LibVersion := '1.0'; ExternalAccessible := 'False'; ExternalVisible := 'False'; ExternalWritable := 'False'; S7_SetPoint := 'False'} : R_TRIG;   // Rising edge of infeeding on upper conveyor
      sR_TRIG_LowerOutfeedRunning {InstructionName := 'R_TRIG'; LibVersion := '1.0'; ExternalAccessible := 'False'; ExternalVisible := 'False'; ExternalWritable := 'False'; S7_SetPoint := 'False'} : R_TRIG;   // Rising edge of outfeeding on lower conveyor
      sR_TRIG_UpperOutfeedRunning {InstructionName := 'R_TRIG'; LibVersion := '1.0'; ExternalAccessible := 'False'; ExternalVisible := 'False'; ExternalWritable := 'False'; S7_SetPoint := 'False'} : R_TRIG;   // Rising edge of outfeeding on upper conveyor
      sR_TRIG_LowerOutfeed {InstructionName := 'R_TRIG'; LibVersion := '1.0'; ExternalAccessible := 'False'; ExternalVisible := 'False'; ExternalWritable := 'False'; S7_SetPoint := 'False'} : R_TRIG;   // Rising edge of outfeed mode on lower conveyor
      sR_TRIG_UpperOutfeed {InstructionName := 'R_TRIG'; LibVersion := '1.0'; ExternalAccessible := 'False'; ExternalVisible := 'False'; ExternalWritable := 'False'; S7_SetPoint := 'False'} : R_TRIG;   // Rising edge of outfeed mode on upper conveyor
      sR_TRIG_AirPressureFault {InstructionName := 'R_TRIG'; LibVersion := '1.0'; ExternalAccessible := 'False'; ExternalVisible := 'False'; ExternalWritable := 'False'; S7_SetPoint := 'False'} : R_TRIG;   // Rising edge of air pressure fault
      sR_TRIG_DivertUpError {InstructionName := 'R_TRIG'; LibVersion := '1.0'; ExternalAccessible := 'False'; ExternalVisible := 'False'; ExternalWritable := 'False'; S7_SetPoint := 'False'} : R_TRIG;   // Rising edge of divert up error
      sR_TRIG_DivertDownError {InstructionName := 'R_TRIG'; LibVersion := '1.0'; ExternalAccessible := 'False'; ExternalVisible := 'False'; ExternalWritable := 'False'; S7_SetPoint := 'False'} : R_TRIG;   // Rising edge of divert down error
      sR_TRIG_PECInfeedA {InstructionName := 'R_TRIG'; LibVersion := '1.0'; ExternalAccessible := 'False'; ExternalVisible := 'False'; ExternalWritable := 'False'; S7_SetPoint := 'False'} : R_TRIG;   // Rising edge on A infeed PEC
      sR_TRIG_PECInfeedB {InstructionName := 'R_TRIG'; LibVersion := '1.0'; ExternalAccessible := 'False'; ExternalVisible := 'False'; ExternalWritable := 'False'; S7_SetPoint := 'False'} : R_TRIG;   // Rising edge on B infeed PEC
      sR_TRIG_PECInfeedC {InstructionName := 'R_TRIG'; LibVersion := '1.0'; ExternalAccessible := 'False'; ExternalVisible := 'False'; ExternalWritable := 'False'; S7_SetPoint := 'False'} : R_TRIG;   // Rising edge on C infeed PEC
      sR_TRIG_PECInfeedD {InstructionName := 'R_TRIG'; LibVersion := '1.0'; ExternalAccessible := 'False'; ExternalVisible := 'False'; ExternalWritable := 'False'; S7_SetPoint := 'False'} : R_TRIG;   // Rising edge on D infeed PEC
      sR_TRIG_LowerInfeedDone {InstructionName := 'R_TRIG'; LibVersion := '1.0'; ExternalAccessible := 'False'; ExternalVisible := 'False'; ExternalWritable := 'False'; S7_SetPoint := 'False'} : R_TRIG;   // Rising edge lower infeed done
      sR_TRIG_UpperInfeedDone {InstructionName := 'R_TRIG'; LibVersion := '1.0'; ExternalAccessible := 'False'; ExternalVisible := 'False'; ExternalWritable := 'False'; S7_SetPoint := 'False'} : R_TRIG;   // Rising edge upper infeed done
   END_VAR
   VAR RETAIN
      si_Step { ExternalAccessible := 'False'; ExternalVisible := 'False'; ExternalWritable := 'False'} : Int;   // Active step number
      si_Conveyor { ExternalAccessible := 'False'; ExternalVisible := 'False'; ExternalWritable := 'False'} : Int;   // Active infeed
   END_VAR
   VAR
      si_LoopArrayCount { ExternalAccessible := 'False'; ExternalVisible := 'False'; ExternalWritable := 'False'} : Int;   // Counter for loop
   END_VAR
   VAR RETAIN
      si_Destination { ExternalAccessible := 'False'; ExternalVisible := 'False'; ExternalWritable := 'False'} : Int;   // Destionation for the product
      si_LowerInfeedDistance { ExternalAccessible := 'False'; ExternalVisible := 'False'; ExternalWritable := 'False'} : Int;   // Counter to receive product on lower conveyor
      si_UpperInfeedDistance { ExternalAccessible := 'False'; ExternalVisible := 'False'; ExternalWritable := 'False'} : Int;   // Counter to receive product on upper conveyor
      si_LowerOutfeedDistance { ExternalAccessible := 'False'; ExternalVisible := 'False'; ExternalWritable := 'False'} : Int;   // Counter to send product from lower conveyor
      si_UpperOutfeedDistance { ExternalAccessible := 'False'; ExternalVisible := 'False'; ExternalWritable := 'False'} : Int;   // Counter to send product from upper conveyor
      sx_PECFiltered { ExternalAccessible := 'False'; ExternalVisible := 'False'; ExternalWritable := 'False'} : Bool;   // Signal filtered with on and off delay
      sx_Active { ExternalAccessible := 'False'; ExternalVisible := 'False'; ExternalWritable := 'False'} : Bool;   // Device sequence is activated for parcel
      sx_DataReceived { ExternalAccessible := 'False'; ExternalVisible := 'False'; ExternalWritable := 'False'} : Bool;   // Destination data is received
      sx_InfeedCHK { ExternalAccessible := 'False'; ExternalVisible := 'False'; ExternalWritable := 'False'} : Bool;   // Step Infeed check
      sx_UpDown { ExternalAccessible := 'False'; ExternalVisible := 'False'; ExternalWritable := 'False'} : Bool;   // Step determine go up or down (wait for destination)
      sx_MoveSectionUpinfeed { ExternalAccessible := 'False'; ExternalVisible := 'False'; ExternalWritable := 'False'} : Bool;   // Step move device to upper position
      sx_MoveSectionUpOutfeed { ExternalAccessible := 'False'; ExternalVisible := 'False'; ExternalWritable := 'False'} : Bool;   // Step move device to upper position
      sx_MoveSectionUpEnd { ExternalAccessible := 'False'; ExternalVisible := 'False'; ExternalWritable := 'False'} : Bool;   // Step move device to upper position
      sx_MoveSectionDownInfeed { ExternalAccessible := 'False'; ExternalVisible := 'False'; ExternalWritable := 'False'} : Bool;   // Step move device to lower position
      sx_MoveSectionDownOutfeed { ExternalAccessible := 'False'; ExternalVisible := 'False'; ExternalWritable := 'False'} : Bool;   // Step move device to lower position
      sx_MoveSectiondownEnd { ExternalAccessible := 'False'; ExternalVisible := 'False'; ExternalWritable := 'False'} : Bool;   // Step move device to lower position
      sx_UpperTransportIn { ExternalAccessible := 'False'; ExternalVisible := 'False'; ExternalWritable := 'False'} : Bool;   // Step transport is activated
      sx_UpperTransportOut { ExternalAccessible := 'False'; ExternalVisible := 'False'; ExternalWritable := 'False'} : Bool;   // Step transport is activated
      sx_LowerTransportIn { ExternalAccessible := 'False'; ExternalVisible := 'False'; ExternalWritable := 'False'} : Bool;   // Step transport is activated
      sx_LowerTransportOut { ExternalAccessible := 'False'; ExternalVisible := 'False'; ExternalWritable := 'False'} : Bool;   // Step transport is activated
      sx_LowerRTR { ExternalAccessible := 'False'; ExternalVisible := 'False'; ExternalWritable := 'False'} : Bool;   // RTR signal to lower level
      sx_UpperRTR { ExternalAccessible := 'False'; ExternalVisible := 'False'; ExternalWritable := 'False'} : Bool;   // RTR signal to upper level
   END_VAR
   VAR
      sx_Ready { ExternalAccessible := 'False'; ExternalVisible := 'False'; ExternalWritable := 'False'} : Bool;   // Conveyor Ready to operate in Automatic mode
      sx_AutomaticActive { ExternalAccessible := 'False'; ExternalVisible := 'False'; ExternalWritable := 'False'} : Bool;   // Running in automatic
      sx_PreStartManual { ExternalAccessible := 'False'; ExternalVisible := 'False'; ExternalWritable := 'False'} : Bool;   // Pre conditions to run conveyor in manual mode
      sx_ManualModeActive { ExternalAccessible := 'False'; ExternalVisible := 'False'; ExternalWritable := 'False'} : Bool;   // Manual mode active
      sx_ManualRunning { ExternalAccessible := 'False'; ExternalVisible := 'False'; ExternalWritable := 'False'} : Bool;   // Device running in manual mode
      sx_ManualGoUp { ExternalAccessible := 'False'; ExternalVisible := 'False'; ExternalWritable := 'False'} : Bool;   // Manual control go Up
      sx_ManualGoDown { ExternalAccessible := 'False'; ExternalVisible := 'False'; ExternalWritable := 'False'} : Bool;   // Manual control go down
      sx_ManUP { ExternalAccessible := 'False'; ExternalVisible := 'False'; ExternalWritable := 'False'} : Bool;   // Auxiliary bit for manual up possition
      sx_ManDown { ExternalAccessible := 'False'; ExternalVisible := 'False'; ExternalWritable := 'False'} : Bool;   // Auxiliary bit for manual down possition
   END_VAR
   VAR RETAIN
      sx_DestinationA { ExternalAccessible := 'False'; ExternalVisible := 'False'; ExternalWritable := 'False'} : Bool;   // Destination is output A
      sx_DestinationB { ExternalAccessible := 'False'; ExternalVisible := 'False'; ExternalWritable := 'False'} : Bool;   // Destination is output B
      sx_DestinationC { ExternalAccessible := 'False'; ExternalVisible := 'False'; ExternalWritable := 'False'} : Bool;   // Destination is output C
      sx_DestinationD { ExternalAccessible := 'False'; ExternalVisible := 'False'; ExternalWritable := 'False'} : Bool;   // Destination is output D
   END_VAR
   VAR
      sx_DivertUpRunTimeErr { ExternalAccessible := 'False'; ExternalVisible := 'False'; ExternalWritable := 'False'} : Bool;   // It is taking too long to move divert up
      sx_DivertDownRunTimeErr { ExternalAccessible := 'False'; ExternalVisible := 'False'; ExternalWritable := 'False'} : Bool;   // It is taking too long to move divert down
      sx_ReactivateA { ExternalAccessible := 'False'; ExternalVisible := 'False'; ExternalWritable := 'False'} : Bool;   // Reactivate conveyor A bit
      sx_ReactivateB { ExternalAccessible := 'False'; ExternalVisible := 'False'; ExternalWritable := 'False'} : Bool;   // Reactivate conveyor B bit
      sx_ReactivateC { ExternalAccessible := 'False'; ExternalVisible := 'False'; ExternalWritable := 'False'} : Bool;   // Reactivate conveyor C bit
      sx_ReactivateD { ExternalAccessible := 'False'; ExternalVisible := 'False'; ExternalWritable := 'False'} : Bool;   // Reactivate conveyor D bit
   END_VAR
   VAR RETAIN
      sx_SectionDown { ExternalAccessible := 'False'; ExternalVisible := 'False'; ExternalWritable := 'False'} : Bool;   // Section down bit
      sx_SectionUp { ExternalAccessible := 'False'; ExternalVisible := 'False'; ExternalWritable := 'False'} : Bool;   // Section up bit
      sx_ProductReceivedDown { ExternalAccessible := 'False'; ExternalVisible := 'False'; ExternalWritable := 'False'} : Bool;   // Product received on lower conveyor
      sx_ProductSentDown { ExternalAccessible := 'False'; ExternalVisible := 'False'; ExternalWritable := 'False'} : Bool;   // Product sent from lower conveyor
      sx_ProductSentUp { ExternalAccessible := 'False'; ExternalVisible := 'False'; ExternalWritable := 'False'} : Bool;   // Product sent from upper conveyor
      sx_ProductReceivedUp { ExternalAccessible := 'False'; ExternalVisible := 'False'; ExternalWritable := 'False'} : Bool;   // Product received on upper conveyor
      sx_ReverseUpper { ExternalAccessible := 'False'; ExternalVisible := 'False'; ExternalWritable := 'False'} : Bool;   // Upper conveyor direction 0 - normal 1 - reverse
      sx_ReverseLower { ExternalAccessible := 'False'; ExternalVisible := 'False'; ExternalWritable := 'False'} : Bool;   // Lower conveyor direction 0 - normal 1 - reverse
      sx_ServoInfeed { ExternalAccessible := 'False'; ExternalVisible := 'False'; ExternalWritable := 'False'} : Bool;   // Infeed base on servo position
      sx_DisplacementInfeed { ExternalAccessible := 'False'; ExternalVisible := 'False'; ExternalWritable := 'False'} : Bool;   // Infeed base on displacement
   END_VAR
   VAR
      sx_TrigPECInfeedA { ExternalAccessible := 'False'; ExternalVisible := 'False'; ExternalWritable := 'False'} : Bool;   // Infeed A released product
      sx_TrigPECInfeedB { ExternalAccessible := 'False'; ExternalVisible := 'False'; ExternalWritable := 'False'} : Bool;   // Infeed B released product
      sx_TrigPECInfeedC { ExternalAccessible := 'False'; ExternalVisible := 'False'; ExternalWritable := 'False'} : Bool;   // Infeed C released product
      sx_TrigPECInfeedD { ExternalAccessible := 'False'; ExternalVisible := 'False'; ExternalWritable := 'False'} : Bool;   // Infeed D released product
      sx_BladeStopEoSControl { ExternalAccessible := 'False'; ExternalVisible := 'False'; ExternalWritable := 'False'} : Bool;   // TRUE when blade stop should go up
      sx_BladeStopBoSControl { ExternalAccessible := 'False'; ExternalVisible := 'False'; ExternalWritable := 'False'} : Bool;   // TRUE when blade stop should go up
      sx_BladeStopUpRunTimeErr { ExternalAccessible := 'False'; ExternalVisible := 'False'; ExternalWritable := 'False'} : Bool;   // It is taking too long for blade stop to move up
      sx_BladeStopDownRunTimeErr { ExternalAccessible := 'False'; ExternalVisible := 'False'; ExternalWritable := 'False'} : Bool;   // It is taking too long for blade stop to move down
   END_VAR

   VAR_TEMP
      tUDT_ConveyorCommandUpper : "UDT_ConveyorCommand";   // Upper conveyor command structure
      tUDT_HMIStatus : "UDT_ConveyorStatus";   // Temporary conveyor hmi status
      tUDT_CommonStatus : "UDT_CommonStatus";   // Temporary conveyor common status
      tUDT_ConveyorStatistics : "UDT_ConveyorStatistics";   // Temporary conveyor statistics
      tUDT_ConveyorInterface : "UDT_ConveyorInterface";   // Temporary conveyor interface
      tx_LowerConveyorRunFwd : Bool;   // Run forward signal for lower conveyor
      tx_UpperConveyorRunFwd : Bool;   // Run backward signal for lower conveyor
      tx_LowerConveyorRunRvs : Bool;   // Run forward signal for upper conveyor
      tx_UpperConveyorRunRvs : Bool;   // Run backwardsignal for upper conveyor
   END_VAR

   VAR CONSTANT
      ci_FiFoLength : Int := 10;   // Fifo length
      ci_ConveyorA : Int := 1;   // Conveyor A is Infeeding
      ci_ConveyorB : Int := 2;   // Conveyor B is Infeeding
      ci_ConveyorC : Int := 3;   // Conveyor C is Infeeding
      ci_ConveyorD : Int := 4;   // Conveyor D is Infeeding
      ci_DefaultPositionUp : Int := 1;
      ci_DefaultPositiondown : Int;
   END_VAR


BEGIN
	(*
	----------------------------------------------------------------------------------------

	Version history:
	Date        | Version   | Author        | Remark
	----------------------------------------------------------------------------------------
	18/10/2023  | 1.0       | F.Baten       | Initial version
	07/11/2023  | 1.1       | K. Pokorski   | Review and tests.
	                                        | Add infeed timeout and infeed reactivation functionality.
	                                        | Fix inserting GIN number to Handshake during outfeed
	                                        | Fix hold control for upper and lower belt of transfer
	                                        | Add reset of RTR when sequence if over
	                                        | Increase length of filling tracking with 0 when outfeed transfer starts
	                                        | Add 4 different destinations input for every infeed separately
	                                        | Unused variables clearing
	                                        | Disable sending RTS because of reverse direction problem and fake FIFO reservations
	02/02/2024  | 1.2       | K.Pokorski    | Add FB conveyor inside RAT block and make code clear and commented
	04/04/2024  | 1.3       | S.Nieswiec    | Newest version from Kamil Pokorski
	08/04/2024  | 1.4       | R. Pieczonka  | Changed writing pneumatic outputs in Region 8.1 due to the valve being monostable
	06/05/2024  | 1.5       | K. Pokorski   | Changed condition for tracking transition
	                                        | Add 4 direction infeed tracking and change condition to track product tail base on infeed PEC
	                                        | Correct product GIN transition
	                                        | Add configuration to disable PEC product controlling
	10/05/2024  | 1.6       | K. Pokorski   | Add outfeed based on displacement
	31/05/2024  | 1.7       | K. Pokorski   | Add positioning infeed control
	28/08/2024  | 1.8       | J.Majer       | Added BoS blade stop, added valve status input interface, removed blade stop position monitoring in RAT block, replaced integers with constants for destination

	*)

	(*
	    From A to B product is transported via rollers
	    From C to D product is transported via pop up belt strips

	                        |             |
	                        |             |
	                        | Conveyor B  |
	                        |      /\     |
	                        |      |      |
	                        |      |      |
	                        |      \/     |
	 _______________________--------------- ________________________
	                        |               |
	                        |               |
	   Conveyor D <-->      |      RAT      |  Conveyor C <-->
	                        |               |
	                        |               |
	 _______________________|               |________________________
	                         ---------------
	                        |      /\      |
	                        |      |       |
	                        |      |       |
	                        |      \/      |
	                        |  Conveyor A  |
	                        |              |
	                        |              |

	*)
	REGION 1 - Initial

	    REGION 1.1 - Triggers

	        // Rising edge trigger manual mode
	        #sR_TRIG_ManualMode(CLK := #iqUDT_RATCommand.ManualMode
	                            OR #iqUDT_EquipmentControl.Command.ManualMode
	                            OR #iqUDT_ConveyorCommand.ManualMode);

	        // Falling edge trigger manual mode
	        #sF_TRIG_ManualMode(CLK := #iqUDT_RATCommand.ManualMode
	                            OR #iqUDT_EquipmentControl.Command.ManualMode
	                            OR #iqUDT_ConveyorCommand.ManualMode);

	        // Rising edge trigger to start in manual mode
	        #sR_TRIG_ManualGoUp(CLK := #iqUDT_RATCommand.ManualUp);

	        // Rising edge trigger manual mode jog
	        #sR_TRIG_ManualGoDown(CLK := #iqUDT_RATCommand.ManualDown);

	        // Rising edge PEC outfeed
	        #sR_TRIG_PecOutfeed(CLK := #sx_PECFiltered);

	        // Infeed conveyor is ready to send
	        #sR_TRIG_ReceiveRequestConveyorA(CLK := (#ix_ExternalReceiveRequestA) AND #ix_ConveyorAAuto);
	        #sR_TRIG_ReceiveRequestConveyorB(CLK := (#ix_ExternalReceiveRequestB) AND #ix_ConveyorBAuto);
	        #sR_TRIG_ReceiveRequestConveyorC(CLK := (#ix_ExternalReceiveRequestC) AND #ix_ConveyorCAuto);
	        #sR_TRIG_ReceiveRequestConveyorD(CLK := (#ix_ExternalReceiveRequestD) AND #ix_ConveyorDAuto);

	        // Rising edge infeed on lower conveyor started
	        #sR_TRIG_LowerInfeed(CLK := #sx_LowerTransportIn);

	        // Rising edge infeed on upper conveyor started
	        #sR_TRIG_UpperInfeed(CLK := #sx_UpperTransportIn);

	        // Rising edge outfeed on lower conveyor started
	        #sR_TRIG_LowerOutfeed(CLK := #sx_LowerTransportOut);

	        // Rising edge outfeed on upper conveyor started
	        #sR_TRIG_UpperOutfeed(CLK := #sx_UpperTransportOut);

	        // Rising edge outfeed on lower conveyor when it's running
	        #sR_TRIG_LowerOutfeedRunning(CLK := #iqUDT_LowerConveyorInterface.ActualSpeed <> 0 AND #sx_LowerTransportOut);

	        // Rising edge outfeed on upper conveyor when it's running
	        #sR_TRIG_UpperOutfeedRunning(CLK := #iqUDT_UpperConveyorInterface.ActualSpeed <> 0 AND #sx_UpperTransportOut);

	        //Rising edge air pressure error occured
	        #sR_TRIG_AirPressureFault(CLK := #sUDT_HMIStatus.Specific.ErrAirpressureNotOk);

	        // Rising edge divert up operation timeout
	        #sR_TRIG_DivertUpError(CLK := #sx_DivertUpRunTimeErr);

	        // Rising edge divert down operation timeout
	        #sR_TRIG_DivertDownError(CLK := #sx_DivertDownRunTimeErr);

	        // Rising edge of Infeed A photoeye
	        #sR_TRIG_PECInfeedA(CLK := #ix_PECInfeedA);

	        // Rising edge of Infeed B photoeye
	        #sR_TRIG_PECInfeedB(CLK := #ix_PECInfeedB);

	        // Rising edge of Infeed C photoeye
	        #sR_TRIG_PECInfeedC(CLK := #ix_PECInfeedC);

	        // Rising edge of Infeed D photoeye
	        #sR_TRIG_PECInfeedD(CLK := #ix_PECInfeedD);

	        // Rising edge lower servo positioning finished
	        #sR_TRIG_LowerInfeedDone(CLK := #iqUDT_RATPositioning.Lower.Done);

	        // Rising edge upper servo positioning finished
	        #sR_TRIG_UpperInfeedDone(CLK := #iqUDT_RATPositioning.Upper.Done);

	    END_REGION

	    REGION 1.2 - Timers

	        // Delay photoeye signal for operation purposes
	        #sFB_PECOnOffDelay(iudi_OnDelayTime := #iUDT_Configuration.OutfeedTimeDelay,
	                           iudi_OffDelayTime := #iUDT_Configuration.InfeedTimeDelay,
	                           ix_SignalToDelay := #ix_PEC,
	                           ix_Enable := TRUE,
	                           qx_DelayedSignal => #sx_PECFiltered);

	        // Monitor upward movement and generate an error when time is exceeded
	        #sFB_SectionUpMonitor(iudi_OnDelayTime := #iUDT_Configuration.SectionUpMonitoringTime,
	                              ix_SignalToDelay := #sx_AutomaticActive
	                              AND #sx_SectionUp
	                              AND NOT #ix_SectionIsUp,
	                              ix_Enable := TRUE,
	                              qx_DelayedSignal => #sx_DivertUpRunTimeErr);

	        // Monitor downward movement and generate an error when time is exceeded
	        #sFB_SectionDownMonitor(iudi_OnDelayTime := #iUDT_Configuration.SectionDownMonitoringTime,
	                                ix_SignalToDelay := #sx_AutomaticActive
	                                AND #sx_SectionDown
	                                AND NOT #ix_SectionIsDown,
	                                ix_Enable := TRUE,
	                                qx_DelayedSignal => #sx_DivertDownRunTimeErr);

	    END_REGION

	    REGION 1.3 - Initialization

	        #iqUDT_RATPositioning.Lower.ResetPosition := FALSE;
	        #iqUDT_RATPositioning.Upper.ResetPosition := FALSE;

	    END_REGION

	END_REGION

	REGION 2 - Error / warning

	    REGION 2.1 - Reset errors

	        IF #iqUDT_EquipmentControl.Command.Reset                        // Reset command received
	        THEN
	            #sUDT_HMIStatus.Specific.ErrRuntime := FALSE;               // reset movement timeout error
	            #sUDT_HMIStatus.Specific.ErrAirpressureNotOk := FALSE;      // reset airpressure error
	        END_IF;

	    END_REGION

	    REGION 2.2 - Set errors

	        // Runtime delay error
	        IF #sx_DivertUpRunTimeErr                                       // It took too long to move up
	            OR #sx_DivertDownRunTimeErr                                 // It took too long to move down
	        THEN
	            #sUDT_HMIStatus.Specific.ErrRuntime := TRUE;                // Set error runtime error
	        END_IF;

	        // Airpressure not ok
	        IF (NOT #ix_AirPressureOk                                        // Airpressure is not signalling
	            AND #sx_SectionUp)                                           // If there is request to move up
	        THEN
	            #sUDT_HMIStatus.Specific.ErrAirpressureNotOk := TRUE;       // Set error airpressure
	        END_IF;

	    END_REGION

	    REGION 2.3 - Warning

	        #sUDT_HMIStatus.Specific.WarnAirPressure := NOT #ix_AirPressureOk;  // Airpressure is not signalling

	    END_REGION


	    REGION 2.4 - Common Error

	        #sUDT_CommonStatus.Error := #sUDT_HMIStatus.Specific.ErrRuntime         // Direction verification found the Direction fault, stop the parcel
	        OR #sUDT_HMIStatus.Specific.ErrAirpressureNotOk                         // Upper jam PEC detected WHILE going Up
	        OR #sUDT_HMIStatus.Specific.ErrOverrun                                  // Parcel travelled too far to divert
	        OR #iqUDT_LowerConveyorInterface.InternalErrorPEC                       // Error PEC on lower conveyor
	        OR #iqUDT_UpperConveyorInterface.InternalErrorPEC                       // Error PEC on upper conveyor
	        OR #iqUDT_LowerConveyorInterface.InternalErrorVFD                       // Error lower conveyor VFD
	        OR #iqUDT_UpperConveyorInterface.InternalErrorVFD                       // Error upper conveyor VFD
	        OR #iqUDT_BladeStopEoSInterface.Error                                   // Blade stop EoS has error
	        OR #iqUDT_BladeStopBoSInterface.Error;                                  // Blade stop BoS has error


	    END_REGION

	    REGION 2.5 - Common Warning

	        #sUDT_CommonStatus.Warning := #sUDT_HMIStatus.Specific.WarnAirPressure;   // Airpressure is not signalling

	    END_REGION

	    REGION 2.6 - Common Stopped

	        #sUDT_CommonStatus.Stopped := NOT #sx_Ready OR NOT #sx_AutomaticActive;       //Device is stopped

	    END_REGION

	END_REGION

	REGION 3 - Check conditions to set Equipment ready

	    //Conditions to set bit sx_Ready to operate

	    #sx_Ready := NOT #sUDT_CommonStatus.Error                           // Error present
	    AND #ix_SafetyOk                                                    // Safety signalling OK
	    AND #ix_24vOk                                                       // 24V signalling OK
	    AND #ix_400vOk;                                                     // 400v signalling OK

	END_REGION

	REGION 4 - Stop Equipment

	    // Conditions to stop conveyor
	    IF (#sF_TRIG_Jog.Q                                                  // Trigger when conveyor stops jogging by HMI
	        AND #sx_ManualModeActive)                                       // Manual mode is active

	        OR (NOT #iqUDT_EquipmentControl.Command.AutomaticOn             // Conveyor stops if the bit AutomaticOn from control block is false
	        AND NOT #sx_ManualModeActive)                                   // Manual mode active bit

	        OR (NOT #sx_Ready                                               // Bit conveyor ready to run in automatic mode
	        AND NOT #sx_ManualModeActive)                                   // Manual mode active

	        OR #sR_TRIG_ManualMode.Q                                        // Trigger when manual mode is set on
	        OR #sF_TRIG_ManualMode.Q                                        // Trigger when manual mode is set off

	        OR NOT #ix_SafetyOk                                             // Safety not ok
	    THEN
	        //  Order to stop VFD
	        #iqUDT_LowerConveyorInterface.RunFwd := FALSE;                       // Set false order to VFD run in forward direction
	        #iqUDT_LowerConveyorInterface.RunRvs := FALSE;                       // Set false order to VFD run in reverse direction
	        #iqUDT_UpperConveyorInterface.RunFwd := FALSE;
	        #iqUDT_UpperConveyorInterface.RunRvs := FALSE;
	        #sx_AutomaticActive := FALSE;                                   // Automatic mode is disable
	    END_IF;

	END_REGION

	REGION 5 - Start

	    REGION 5.1 - Set Automatic active

	        // The conditions to set the bit "startReceived" are:
	        // - Divert not in manual mode.
	        // - Divert ready to run.
	        // - Bit AutomaticOn from control block must be on.
	        // - Bit start form control block on.

	        IF #iqUDT_EquipmentControl.Command.Start
	            AND #iqUDT_EquipmentControl.Command.AutomaticOn
	            AND NOT #sx_ManualModeActive
	            AND #sx_Ready
	        THEN
	            #sx_AutomaticActive := TRUE;                                // Diverter active automatic mode
	        END_IF;

	    END_REGION

	    REGION 5.2 - Restart request

	        #iqUDT_EquipmentControl.Request.RestartRequired := NOT #sx_AutomaticActive
	        AND NOT #sx_ManualModeActive
	        AND #sx_Ready;

	    END_REGION

	END_REGION

	REGION 6 - Manual mode

	    REGION 6.1 - Manual mode force disable

	        // Manual mode bits inputs can be reset in case of malfunction
	        IF #iqUDT_EquipmentControl.Command.DisableManualMode
	        THEN
	            #iqUDT_RATCommand.ManualMode := FALSE;
	            #iqUDT_EquipmentControl.Command.ManualMode := False;
	        END_IF;

	    END_REGION

	    REGION 6.2 - Manual mode activation

	        // Manual mode is active if it is active from hmi or by control block
	        #sx_ManualModeActive := #iqUDT_RATCommand.ManualMode
	        OR #iqUDT_EquipmentControl.Command.ManualMode
	        OR #iqUDT_ConveyorCommand.ManualMode;

	    END_REGION

	    REGION 6.3 - Reset manual commands
	        //When the system is not any more in manual mode or when fatal error occurs the HMI commands should be reset
	        IF NOT #ix_SafetyOk                                             // Safety not ok
	            OR NOT #ix_24vOk                                            // 24V error status
	            OR NOT #ix_400vOk                                           // 400V error status
	            OR NOT #ix_HardwareOk                                       // Profinet error status
	            OR NOT #sx_ManualModeActive                                 // Manual mode active
	        THEN
	            #iqUDT_RATCommand.ManualDown := FALSE;                      // Reset movement command
	            #iqUDT_RATCommand.ManualUp := FALSE;                        // Reset movement command
	        END_IF;

	    END_REGION

	    REGION 6.4 - Start/Stop

	        // Pre start conditions to run in manual mode
	        #sx_PreStartManual := #sx_ManualModeActive                      // Manual mode active bit
	        AND #ix_SafetyOk                                                // Safety healthy bit
	        AND #ix_HardwareOk;                                             // Profinet comunication

	        // If manual command is active to one side, first button has to be released to accept new
	        #sx_ManUP := (#sR_TRIG_ManualGoUp.Q AND NOT #sx_ManDown) OR
	        (#sx_ManUP AND #iqUDT_RATCommand.ManualUp);

	        #sx_ManDown := (#sR_TRIG_ManualGoDown.Q AND NOT #sx_ManUP) OR
	        (#sx_ManDown AND #iqUDT_RATCommand.ManualDown);

	        // Do signal request (horn sounding before movement)
	        IF #sx_PreStartManual                                           // Pre start conditions to run in manual mode
	            AND (#sR_TRIG_ManualGoUp.Q AND #sx_ManUP)                  // Trigger when conveyor start running in manual mode
	            OR (#sR_TRIG_ManualGoDown.Q AND #sx_ManDown)
	        THEN

	            #iqUDT_EquipmentControl.Request.SignalingRequest := TRUE;   // Request signaling to control block before conveyor run in manual mode

	        END_IF;

	        // Go up in manual mode
	        #sx_ManualGoUp := #sx_PreStartManual                            // Pre start conditions to run in manual mode
	        AND (NOT #iqUDT_EquipmentControl.Request.SignalingRequest       // Signaling request done
	        OR #sx_ManualRunning)
	        AND #sx_ManUP;
	        ;                                                // Manual mode start TO run

	        // Go down in manual mode
	        #sx_ManualGoDown := #sx_PreStartManual                          // Pre start conditions to run in manual mode
	        AND (NOT #iqUDT_EquipmentControl.Request.SignalingRequest       // Signaling request done
	        OR #sx_ManualRunning)
	        AND #sx_ManDown;                                                // Manual mode start to run

	        #sx_ManualRunning := #sx_ManualGoUp
	        OR #sx_ManualGoDown;

	    END_REGION

	END_REGION

	REGION 7 - Automatic mode
	    REGION 7.1 - Update FiFo
	        FOR #si_LoopArrayCount := 1 TO (#ci_FiFoLength - 1) BY 1 DO                 // Set loop to process
	            IF #sa_FiFo[#si_LoopArrayCount] = 0                                     // Do when actual value is '0'
	            THEN
	                #sa_FiFo[#si_LoopArrayCount] := #sa_FiFo[#si_LoopArrayCount + 1];   // copy next entry to actual
	                #sa_FiFo[#si_LoopArrayCount + 1] := 0;                              // Reset next entry
	            END_IF;
	        END_FOR;
	        // Get double entry out
	        IF #sx_Active                                                               // When Sequence is activated
	        THEN
	            IF (#sa_FiFo[2] <> 0)                                                   // Entry 2 is not equal to '0'
	                AND (#sa_FiFo[2] = #sa_FiFo[3])                                     // Entry 2 is equal to 3
	            THEN
	                #sa_FiFo[3] := 0;                                                   // remove entry 3
	            ELSIF
	                (#sa_FiFo[2] <> 0)                                                  // Entry 2 is not equal to '0'
	                AND (#sa_FiFo[2] = #sa_FiFo[4])                                     // Entry 2 is equal to 4
	            THEN
	                #sa_FiFo[4] := 0;                                                   // Remove entry 4
	            END_IF;
	        END_IF;
	    END_REGION

	    REGION 7.2 - FIFO handling
	        // When an infeed send command it is put in the FiFo then the FiFo is shifted.

	        IF #sR_TRIG_ReceiveRequestConveyorA.Q                                           // Signal received from infeed A
	            OR #sx_ReactivateA                                                          // Reactivate infeed A request
	        THEN
	            #sa_FiFo[#ci_FiFoLength] := 1;                                              // Set last FiFo entry to A

	            FOR #si_LoopArrayCount := 1 TO (#ci_FiFoLength - 1) BY 1 DO                 // Set loop to process
	                IF #sa_FiFo[#si_LoopArrayCount] = 0                                     // Do when actual value is '0'
	                THEN
	                    #sa_FiFo[#si_LoopArrayCount] := #sa_FiFo[#si_LoopArrayCount + 1];   // copy next entry to actual
	                    #sa_FiFo[#si_LoopArrayCount + 1] := 0;                              // Reset next entry
	                END_IF;
	            END_FOR;
	            #sx_ReactivateA := FALSE;                                                   // Clear reactivation bit for conveyor A
	        END_IF;

	        IF #sR_TRIG_ReceiveRequestConveyorB.Q                                           // Signal received from infeed B
	            OR #sx_ReactivateB                                                          // Reactivate infeed B request
	        THEN
	            #sa_FiFo[#ci_FiFoLength] := 2;                                              // Set last FiFo entry to B

	            FOR #si_LoopArrayCount := 1 TO (#ci_FiFoLength - 1) BY 1 DO                 // Set loop to process
	                IF #sa_FiFo[#si_LoopArrayCount] = 0                                     // Do when actual value is '0'
	                THEN
	                    #sa_FiFo[#si_LoopArrayCount] := #sa_FiFo[#si_LoopArrayCount + 1];   // copy next entry to actual
	                    #sa_FiFo[#si_LoopArrayCount + 1] := 0;                              // Reset next entry
	                END_IF;
	            END_FOR;
	            #sx_ReactivateB := FALSE;                                                   // Clear reactivation bit for conveyor B
	        END_IF;

	        IF #sR_TRIG_ReceiveRequestConveyorC.Q                                           // Signal received from infeed C
	            OR #sx_ReactivateC                                                          // Reactivate infeed C request
	        THEN
	            #sa_FiFo[#ci_FiFoLength] := 3;                                              // Set last FiFo entry to C

	            FOR #si_LoopArrayCount := 1 TO (#ci_FiFoLength - 1) BY 1 DO                 // Set loop to process
	                IF #sa_FiFo[#si_LoopArrayCount] = 0                                     // Do when actual value is '0'
	                THEN
	                    #sa_FiFo[#si_LoopArrayCount] := #sa_FiFo[#si_LoopArrayCount + 1];   // copy next entry to actual
	                    #sa_FiFo[#si_LoopArrayCount + 1] := 0;                              // Reset next entry
	                END_IF;
	            END_FOR;
	            #sx_ReactivateC := FALSE;                                                   // Clear reactivation bit for conveyor C
	        END_IF;

	        IF #sR_TRIG_ReceiveRequestConveyorD.Q                                           // Signal received from infeed D
	            OR #sx_ReactivateD                                                          // Reactivate infeed D request
	        THEN
	            #sa_FiFo[#ci_FiFoLength] := 4;                                              // Set last FiFo entry to D

	            FOR #si_LoopArrayCount := 1 TO (#ci_FiFoLength - 1) BY 1 DO                 // Set loop to process
	                IF #sa_FiFo[#si_LoopArrayCount] = 0                                     // Do when actual value is '0'
	                THEN
	                    #sa_FiFo[#si_LoopArrayCount] := #sa_FiFo[#si_LoopArrayCount + 1];   // copy next entry to actual
	                    #sa_FiFo[#si_LoopArrayCount + 1] := 0;                              // Reset next entry
	                END_IF;
	            END_FOR;
	            #sx_ReactivateD := FALSE;                                                   // Clear reactivation bit for conveyor D
	        END_IF;
	    END_REGION

	    REGION 7.3 - Start sequence, infeed conveyor request

	        REGION 7.3.1 - Start sequence, infeed conveyor request
	            // If FiFo has an entry which is matching request, the request is rewarded and the sequence is started
	            IF NOT #sx_Active                                               // Not activated yet
	                AND #sa_FiFo[1] <> 0                                        // There is a request in FiFo 1
	            THEN
	                IF #sa_FiFo[1] = #ci_ConveyorA                              // Conveyor A is infeed
	                    AND #ix_ExternalReceiveRequestA                         // Check if infeed A requested send
	                THEN
	                    #sx_InfeedCHK := TRUE;                                  // Infeed is checked
	                    #si_Conveyor := #ci_ConveyorA;                          // Set active infeed

	                ELSIF #sa_FiFo[1] = #ci_ConveyorB                           // Conveyor B is infeed
	                    AND #ix_ExternalReceiveRequestB                         // Check if infeed B requested send
	                THEN
	                    #sx_InfeedCHK := TRUE;                                  // Infeed is checked
	                    #si_Conveyor := #ci_ConveyorB;                          // Set active infeed

	                ELSIF #sa_FiFo[1] = #ci_ConveyorC                           // Conveyor C is infeed
	                    AND #ix_ExternalReceiveRequestC                         // Check if infeed C requested send
	                THEN
	                    #sx_InfeedCHK := TRUE;                                  // Infeed is checked
	                    #si_Conveyor := #ci_ConveyorC;                          // Set active infeed

	                ELSIF #sa_FiFo[1] = #ci_ConveyorD                           // Conveyor D is infeed
	                    AND #ix_ExternalReceiveRequestD                         // Check if infeed D requested send
	                THEN
	                    #sx_InfeedCHK := TRUE;                                  // Infeed is checked
	                    #si_Conveyor := #ci_ConveyorD;                          // Set active infeed
	                ELSE
	                    #sa_FiFo[1] := 0;                                       // No infeed request was matching
	                END_IF;

	                IF #sx_InfeedCHK                                            // Infeed is checked
	                THEN
	                    #sx_Active := TRUE;                                     // Sequence is started
	                    #sa_FiFo[1] := 0;                                       // Reset entry D
	                    #si_Step := 1;                                          // Set step number for diagnostic purposes
	                END_IF;
	            END_IF;
	        END_REGION

	        REGION 7.3.2 Receiving destination from input
	            IF NOT #sx_DataReceived                                                                                             // Data is not yet received
	                AND (#sx_LowerTransportIn AND (#sR_TRIG_PECInfeedA.Q OR #sR_TRIG_PECInfeedB.Q))                                 // Try to get data during lower infeed
	                OR (#sx_UpperTransportIn AND (#sR_TRIG_PECInfeedC.Q OR #sR_TRIG_PECInfeedD.Q))                                  // Try to get data during upper infeed
	                OR #sx_UpDown                                                                                                   // Infeed transport or waiting for data
	            THEN
	                IF #si_Conveyor = #ci_ConveyorA
	                THEN                                                                                        // Search destination for product from Conveyor A
	                    IF #ii_DestinationA <> 0
	                    THEN                                                                               // Destination is forced from output
	                        #si_Destination := #ii_DestinationA;
	                    ELSIF #sUDT_HandshakeBuffer.GIN <> 0
	                    THEN
	                        IF "DB_GIN".GIN[#sUDT_HandshakeBuffer.GIN].General.Destination[0] <> 0                                  // Destination is not forced from output and GIN is detected
	                        THEN
	                            #si_Destination := DINT_TO_INT("DB_GIN".GIN[#sUDT_HandshakeBuffer.GIN].General.Destination[0]);     // Divert product to the GIN destination
	                        END_IF;
	                    END_IF;

	                ELSIF #si_Conveyor = #ci_ConveyorB
	                THEN                                                                                     // Search destination for product from Conveyor B
	                    IF #ii_DestinationB <> 0
	                    THEN                                                                               // Destination is forced from output
	                        #si_Destination := #ii_DestinationB;
	                    ELSIF #sUDT_HandshakeBuffer.GIN <> 0
	                    THEN
	                        IF "DB_GIN".GIN[#sUDT_HandshakeBuffer.GIN].General.Destination[0] <> 0                                  // Destination is not forced from output and GIN is detected
	                        THEN
	                            #si_Destination := DINT_TO_INT("DB_GIN".GIN[#sUDT_HandshakeBuffer.GIN].General.Destination[0]);     // Divert product to the GIN destination
	                        END_IF;
	                    END_IF;
	                ELSIF #si_Conveyor = #ci_ConveyorC
	                THEN                                                                                     // Search destination for product from Conveyor C
	                    IF #ii_DestinationC <> 0
	                    THEN                                                                               // Destination is forced from output
	                        #si_Destination := #ii_DestinationC;
	                    ELSIF #sUDT_HandshakeBuffer.GIN <> 0
	                    THEN
	                        IF "DB_GIN".GIN[#sUDT_HandshakeBuffer.GIN].General.Destination[0] <> 0                                  // Destination is not forced from output and GIN is detected
	                        THEN
	                            #si_Destination := DINT_TO_INT("DB_GIN".GIN[#sUDT_HandshakeBuffer.GIN].General.Destination[0]);     // Divert product to the GIN destination
	                        END_IF;
	                    END_IF;
	                ELSIF #si_Conveyor = #ci_ConveyorD
	                THEN                                                                                     // Search destination for product from Conveyor D
	                    IF #ii_DestinationD <> 0
	                    THEN                                                                               // Destination is forced from output
	                        #si_Destination := #ii_DestinationD;
	                    ELSIF #sUDT_HandshakeBuffer.GIN <> 0
	                    THEN
	                        IF "DB_GIN".GIN[#sUDT_HandshakeBuffer.GIN].General.Destination[0] <> 0                                  // Destination is not forced from output and GIN is detected
	                        THEN
	                            #si_Destination := DINT_TO_INT("DB_GIN".GIN[#sUDT_HandshakeBuffer.GIN].General.Destination[0]);     // Divert product to the GIN destination
	                        END_IF;
	                    END_IF;
	                END_IF;

	                IF #si_Destination > 0
	                THEN                                     // Destination is not '0'
	                    #sx_DataReceived := TRUE;                                   // Data is valid
	                END_IF;


	                // Destination received, set the appropriate bit

	                #sx_DestinationA := #sx_DataReceived AND (#iUDT_Configuration.ConveyorADestination = #si_Destination);
	                #sx_DestinationB := #sx_DataReceived AND (#iUDT_Configuration.ConveyorBDestination = #si_Destination);
	                #sx_DestinationC := #sx_DataReceived AND (#iUDT_Configuration.ConveyorCDestination = #si_Destination);
	                #sx_DestinationD := #sx_DataReceived AND (#iUDT_Configuration.ConveyorDDestination = #si_Destination);


	                // If destination is not configured then go to default destination
	                IF NOT #sx_DestinationA AND NOT #sx_DestinationB AND NOT #sx_DestinationC AND NOT #sx_DestinationD
	                THEN

	                    IF #iUDT_Configuration.DefaultDestination = #ci_ConveyorA
	                    THEN
	                        #sx_DestinationA := TRUE;
	                        #sx_DataReceived := TRUE;
	                    ELSIF #iUDT_Configuration.DefaultDestination = #ci_ConveyorB
	                    THEN
	                        #sx_DestinationB := TRUE;
	                        #sx_DataReceived := TRUE;
	                    ELSIF #iUDT_Configuration.DefaultDestination = #ci_ConveyorC
	                    THEN
	                        #sx_DestinationC := TRUE;
	                        #sx_DataReceived := TRUE;
	                    ELSIF #iUDT_Configuration.DefaultDestination = #ci_ConveyorD
	                    THEN
	                        #sx_DestinationD := TRUE;
	                        #sx_DataReceived := TRUE;
	                    END_IF;
	                END_IF;
	            END_IF;

	        END_REGION

	        REGION 7.3.3 - Lower infeed product tracking

	            //Trigger from PEC-infeed A
	            IF #sR_TRIG_PECInfeedA.Q
	                AND #si_Conveyor = #ci_ConveyorA
	                AND #sx_LowerTransportIn
	                AND NOT #sx_ServoInfeed
	                AND NOT #sx_DisplacementInfeed
	            THEN
	                #sx_TrigPECInfeedA := TRUE;
	            END_IF;

	            //Waiting for new postion from input, then setting end position
	            IF #sx_TrigPECInfeedA
	                AND #iqUDT_RATPositioning.Lower.StartPositionA <> 0
	                AND ((#sx_DataReceived
	                AND NOT #sx_DestinationB)
	                OR NOT #sx_DataReceived)
	            THEN
	                #sx_ServoInfeed := TRUE;
	                #iqUDT_RATPositioning.Lower.EndPosition := #iqUDT_RATPositioning.Lower.StartPositionA + #iUDT_Configuration.InfeedADistance;
	                #sx_TrigPECInfeedA := FALSE;
	                #iqUDT_RATPositioning.Lower.StartPositionA := 0;
	                #iqUDT_RATPositioning.Lower.PositionRequired := FALSE;
	                #iqUDT_RATPositioning.Lower.Start := TRUE;

	                // If straight destination detected then use displacement mode
	            ELSIF #sx_TrigPECInfeedA
	                AND #sx_DataReceived
	                AND #sx_DestinationB
	            THEN
	                #si_LowerInfeedDistance := ABS(#iUDT_Configuration.InfeedADistance / 10);
	                #sx_TrigPECInfeedA := FALSE;
	                #sx_DisplacementInfeed := TRUE;
	                #iqUDT_RATPositioning.Lower.StartPositionA := 0;
	                #iqUDT_RATPositioning.Lower.PositionRequired := FALSE;
	            END_IF;

	            //Trigger from PEC-infeed B
	            IF #sR_TRIG_PECInfeedB.Q
	                AND #si_Conveyor = #ci_ConveyorB
	                AND #sx_LowerTransportIn
	                AND NOT #sx_ServoInfeed
	                AND NOT #sx_DisplacementInfeed
	            THEN
	                #sx_TrigPECInfeedB := TRUE;
	            END_IF;

	            //Waiting for new postion from input, then setting end position
	            IF #sx_TrigPECInfeedB
	                AND #iqUDT_RATPositioning.Lower.StartPositionB <> 0
	                AND ((#sx_DataReceived
	                AND NOT #sx_DestinationA)
	                OR NOT #sx_DataReceived)
	            THEN
	                #sx_ServoInfeed := TRUE;
	                #iqUDT_RATPositioning.Lower.EndPosition := #iqUDT_RATPositioning.Lower.StartPositionB - #iUDT_Configuration.InfeedBDistance;
	                #sx_TrigPECInfeedB := FALSE;
	                #iqUDT_RATPositioning.Lower.StartPositionB := 0;
	                #iqUDT_RATPositioning.Lower.PositionRequired := FALSE;
	                #iqUDT_RATPositioning.Lower.Start := TRUE;
	                // If straight destination detected then use displacement mode
	            ELSIF #sx_TrigPECInfeedB
	                AND #sx_DataReceived
	                AND #sx_DestinationA
	            THEN
	                #si_LowerInfeedDistance := ABS(#iUDT_Configuration.InfeedBDistance / 10);
	                #sx_TrigPECInfeedB := FALSE;
	                #sx_DisplacementInfeed := TRUE;
	                #iqUDT_RATPositioning.Lower.StartPositionB := 0;
	                #iqUDT_RATPositioning.Lower.PositionRequired := FALSE;
	            END_IF;


	            //If position is reached, set ProductRecived
	            IF #sR_TRIG_LowerInfeedDone.Q
	                AND #sx_ServoInfeed
	            THEN
	                #sx_ProductReceivedDown := TRUE;
	                #iqUDT_RATPositioning.Lower.Start := FALSE;
	            END_IF;

	            // During lower infeeding count distance to end of RAT
	            IF #sx_LowerTransportIn AND
	                #sx_DisplacementInfeed
	                AND NOT #sx_ProductReceivedDown
	            THEN
	                #si_LowerInfeedDistance -= ABS(#iqUDT_LowerConveyorInterface.Displacement);
	                IF #si_LowerInfeedDistance <= 0
	                THEN
	                    #sx_ProductReceivedDown := TRUE;
	                END_IF;
	            END_IF;

	        END_REGION

	        REGION 7.3.4 - Upper infeed product tracking

	            //Trigger from PEC-infeed C
	            IF #sR_TRIG_PECInfeedC.Q
	                AND #si_Conveyor = #ci_ConveyorC
	                AND #sx_UpperTransportIn
	                AND NOT #sx_ServoInfeed
	                AND NOT #sx_DisplacementInfeed
	            THEN
	                #sx_TrigPECInfeedC := TRUE;
	            END_IF;

	            //Waiting for new postion from input, then setting end position
	            IF #sx_TrigPECInfeedC
	                AND #iqUDT_RATPositioning.Upper.StartPositionC <> 0
	                AND ((#sx_DataReceived
	                AND NOT #sx_DestinationD)
	                OR NOT #sx_DataReceived)
	            THEN
	                #sx_ServoInfeed := TRUE;
	                #iqUDT_RATPositioning.Upper.EndPosition := #iqUDT_RATPositioning.Upper.StartPositionC + #iUDT_Configuration.InfeedCDistance;
	                #sx_TrigPECInfeedC := FALSE;
	                #iqUDT_RATPositioning.Upper.StartPositionC := 0;
	                #iqUDT_RATPositioning.Upper.PositionRequired := FALSE;
	                #iqUDT_RATPositioning.Upper.Start := TRUE;
	                // If straight destination detected then use displacement mode
	            ELSIF #sx_TrigPECInfeedC
	                AND #sx_DataReceived
	                AND #sx_DestinationD
	            THEN
	                #si_UpperInfeedDistance := ABS(#iUDT_Configuration.InfeedCDistance / 10);
	                #sx_TrigPECInfeedC := FALSE;
	                #sx_DisplacementInfeed := TRUE;
	                #iqUDT_RATPositioning.Upper.StartPositionC := 0;
	                #iqUDT_RATPositioning.Upper.PositionRequired := FALSE;
	            END_IF;

	            //Trigger from PEC-infeed D
	            IF #sR_TRIG_PECInfeedD.Q
	                AND #si_Conveyor = #ci_ConveyorD
	                AND #sx_UpperTransportIn
	                AND NOT #sx_ServoInfeed
	                AND NOT #sx_DisplacementInfeed
	            THEN
	                #sx_TrigPECInfeedD := TRUE;
	            END_IF;

